// ---- POUs/EL_Terminals/FB_EL3403.TcPOU
(************************************************************************************************)
(*							Beckhoff Automation Poland											*)
(*								FB_EL3403	 v1.0												*)
(*									11.03.2014													*)
(*					Blok funkcyjny obsługujący moduł EL3403										*)
(*			Możliwy zapis energii w module, kasowanie przechowywanych wartosci					*)
(*		Jesli jest wybrany wiecej niz jeden kanal to komenda wykonana zostanie na wszystkich	*)
(*					Zapis ma wyzszy priorytet niz kasowanie										*)
(*							Blok posiada fukcje autozapisu										*)
(*				Komendy wkonywane sa na narastajace zbocze na odpowiednim wejsciu				*)
(*______________________________________________________________________________________________*)
FUNCTION_BLOCK FB_EL3403
VAR_INPUT
	sNetId					:	T_AmsNetId;							(* AMS Net ID of EtherCAT Master *)
	nSlaveAddr				:	UINT;
	bStoreCh1				:	BOOL;
	bStoreCh2				:	BOOL;
	bStoreCh3				:	BOOL;
	bStoreAll				:	BOOL;
	bAutoStore				:	BOOL;
	bDeleteCh1				:	BOOL;
	bDeleteCh2				:	BOOL;
	bDeleteCh3				:	BOOL;
	bDeleteAll				:	BOOL;
END_VAR
VAR_OUTPUT
	bBusy					:	BOOL;
	bError					:	BOOL;
	nErrorID				:	UDINT;
	bMissingZeroCrossingA 	AT %I*: 	BOOL;
	bMissingZeroCrossingB 	AT %I*:		BOOL;
	bMissingZeroCrossingC 	AT %I*: 	BOOL;
	bPhaseSequenceError		AT %I*: 	BOOL;
	rCurrent1				:	REAL; (* Unit 1 A *)
	rCurrent2				: 	REAL; (* Unit 1 A *)
	rCurrent3				: 	REAL; (* Unit 1 A *)
	rVoltage1				: 	REAL; (* Unit 1 V *)
	rVoltage2				: 	REAL; (* Unit 1 V *)
	rVoltage3				: 	REAL; (* Unit 1 V *)
	rActivePower1			: 	REAL; (* Unit 1 W *)
	rActivePower2			: 	REAL; (* Unit 1 W *)
	rActivePower3			: 	REAL; (* Unit 1 W *)
	rApparentPower1			: 	REAL; (* Unit 1 VA *)
	rApparentPower2			:	REAL; (* Unit 1 VA *)
	rApparentPower3			:	REAL; (* Unit 1 VA *)
	rReactivePower1			:	REAL; (* Unit 1 VAR *)
	rReactivePower2			:	REAL; (* Unit 1 VAR *)
	rReactivePower3			:	REAL; (* Unit 1 VAR *)
	rEnergy1				: 	REAL; (* Unit 1 Wh *)
	rEnergy2				:	REAL; (* Unit 1 Wh *)
	rEnergy3				: 	REAL; (* Unit 1 Wh *)
	rCosPhi1				: 	REAL; (* Unit 1 *)
	rCosPhi2				: 	REAL; (* Unit 1 *)
	rCosPhi3				: 	REAL; (* Unit 1 *)
	rFrequency1				: 	REAL; (* Unit 1 Hz *)
	rFrequency2				: 	REAL; (* Unit 1 Hz *)
	rFrequency3				: 	REAL; (* Unit 1 Hz *)
	rEnergyNegative1		: 	REAL; (* Unit 1 Wh *)
	rEnergyNegative2		: 	REAL; (* Unit 1 Wh *)
	rEnergyNegative3		: 	REAL; (* Unit 1 Wh *)
END_VAR
VAR
(* I/O *)
	diCurrent1 				AT %I*: DINT;(* Unit 0,000001 A *)
	diCurrent2 				AT %I*: DINT;(* Unit 0,000001 A *)
	diCurrent3 				AT %I*: DINT;(* Unit 0,000001 A *)
	diVoltage1 				AT %I*: DINT;(* Unit 0,0001 V *)
	diVoltage2 				AT %I*: DINT;(* Unit 0,0001 V *)
	diVoltage3 				AT %I*: DINT;(* Unit 0,0001 V *)
	diActivePower1 			AT %I*: DINT;(* Unit 0,01 W *)
	diActivePower2 			AT %I*: DINT;(* Unit 0,01 W *)
	diActivePower3 			AT %I*: DINT;(* Unit 0,01 W *)
	usiIndex1			 	AT %I*: USINT;
	usiIndex2			 	AT %I*: USINT;
	usiIndex3			 	AT %I*: USINT;
	diVariantValue1 		AT %I*: DINT;
	diVariantValue2 		AT %I*: DINT;
	diVariantValue3 		AT %I*: DINT;
	usiIndex1q				AT %Q*: USINT;
	usiIndex2q			 	AT %Q*: USINT;
	usiIndex3q			 	AT %Q*: USINT;
(*Raw Values*)
	diApparentPower1		: DINT; (* Unit 0,01 VA *)
	diApparentPower2		: DINT; (* Unit 0,01 VA *)
	diApparentPower3		: DINT; (* Unit 0,01 VA *)
	diReactivePower1		: DINT; (* Unit 0,01 VAR *)
	diReactivePower2		: DINT; (* Unit 0,01 VAR *)
	diReactivePower3		: DINT; (* Unit 0,01 VAR *)
	diEnergy1				: DINT;(* Unit 0,001 Wh *)
	diEnergy2				: DINT;(* Unit 0,001 Wh *)
	diEnergy3				: DINT;(* Unit 0,001 Wh *)
	diCosPhi1				: DINT;(* Unit 0,001 *)
	diCosPhi2				: DINT;(* Unit 0,001 *)
	diCosPhi3				: DINT;(* Unit 0,001 *)
	diFrequency1			: DINT;(* Unit 0,1 Hz *)
	diFrequency2			: DINT;(* Unit 0,1 Hz *)
	diFrequency3			: DINT;(* Unit 0,1 Hz *)
	diEnergyNegative1		: DINT;(* Unit 0,001 Wh *)
	diEnergyNegative2		: DINT;(* Unit 0,001 Wh *)
	diEnergyNegative3		: DINT;(* Unit 0,001 Wh *)
(* Energy store/delete *)
	fbEcCoeSdoWrite			: FB_EcCoESdoWrite;
	t1						: TON;
	arrRTrigs				: ARRAY [1..9] OF R_TRIG;
	wDataS					: WORD;
	wDataD					: WORD;
	bExecute				: BOOL;
	BStore					: BYTE; (* bit 0 - ch1, 1 - ch2, 3 - ch3, else all *)
	BDelete					: BYTE; (* bit 0 - ch1, 1 - ch2, 3 - ch3, else all *)
	bStoreCommand			: BOOL;
	bDeleteCommand			: BOOL;
	wData					: WORD;
END_VAR
VAR CONSTANT
	nSubIndex				: BYTE				:= 16#01;
	nIndex					: WORD				:= 16#FB00;
	wChannel1				: WORD				:= 16#0100;
	wChannel2				: WORD				:= 16#0200;
	wChannel3				: WORD				:= 16#0300;
	wStore					: WORD				:= 16#0014;
	wDelete					: WORD				:= 16#0004;
	tStoreInterval			: TIME				:= T#15m;
END_VAR

(* Read Variant Variable *)
A_ReadVariantVariable();

(* Scale *)
A_Scale();

(* Energy *)
BStore.0 := bStoreCh1 OR bStoreAll;
BStore.1 := bStoreCh2 OR bStoreAll;
BStore.2 := bStoreCh3 OR bStoreAll;
CASE BStore OF
1:	wDataS := wChannel1 + wStore;
2:	wDataS := wChannel2 + wStore;
4:	wDataS := wChannel3 + wStore;
ELSE
	wDataS := wStore;
END_CASE

BDelete.0 := bDeleteCh1 OR bDeleteAll;
BDelete.1 := bDeleteCh2 OR bDeleteAll;
BDelete.2 := bDeleteCh3 OR bDeleteAll;
CASE BDelete OF
1:	wDataD := wChannel1 + wDelete;
2:	wDataD := wChannel2 + wDelete;
4:	wDataD := wChannel3 + wDelete;
ELSE
	wDataD := wDelete;
END_CASE

t1(IN:= NOT t1.Q AND bAutoStore , PT:= tStoreInterval); (* Auto store *)

arrRTrigs[1](CLK:= bStoreCh1);
arrRTrigs[2](CLK:= bStoreCh2);
arrRTrigs[3](CLK:= bStoreCh3);
arrRTrigs[4](CLK:= bStoreAll);
arrRTrigs[5](CLK:= t1.Q);
arrRTrigs[6](CLK:= bDeleteCh1);
arrRTrigs[7](CLK:= bDeleteCh2);
arrRTrigs[8](CLK:= bDeleteCh3);
arrRTrigs[9](CLK:= bDeleteAll);

bStoreCommand		:= arrRTrigs[1].Q OR arrRTrigs[2].Q OR arrRTrigs[3].Q OR arrRTrigs[4].Q OR arrRTrigs[5].Q;
bDeleteCommand	:= arrRTrigs[6].Q OR arrRTrigs[7].Q OR arrRTrigs[8].Q OR arrRTrigs[9].Q;
wData				:= SEL(bDeleteCommand, wDataS, wDataD);
bExecute			:= bStoreCommand OR bDeleteCommand;




fbEcCoeSdoWrite(
	sNetId:= sNetId,
	nSlaveAddr:= nSlaveAddr,
	nSubIndex:= nSubIndex,
	nIndex:= nIndex,
	pSrcBuf:= ADR(wData),
	cbBufLen:= 2,
	bExecute:= bExecute,
	bBusy=> bBusy,
	bError=> bError,
	nErrId=> nErrorID);

ACTION A_ReadVariantVariable:
CASE usiIndex1 OF
0:
	diApparentPower1 := diVariantValue1;
	usiIndex1q := usiIndex1+1;
1:
	diReactivePower1 := diVariantValue1;
	usiIndex1q := usiIndex1+1;
2:
	diEnergy1 := diVariantValue1;
	usiIndex1q := usiIndex1+1;
3:
	diCosPhi1 := diVariantValue1;
	usiIndex1q := usiIndex1+1;
4:
	diFrequency1 := diVariantValue1;
	usiIndex1q := usiIndex1+1;
5:
	diEnergyNegative1 := diVariantValue1;
	usiIndex1q := usiIndex1+1;
ELSE
	usiIndex1q := 0;
END_CASE

CASE usiIndex2 OF
0:
	diApparentPower2 := diVariantValue2;
	usiIndex2q := usiIndex2+1;
1:
	diReactivePower2 := diVariantValue2;
	usiIndex2q := usiIndex2+1;
2:
	diEnergy2 := diVariantValue2;
	usiIndex2q := usiIndex2+1;
3:
	diCosPhi2 := diVariantValue2;
	usiIndex2q := usiIndex2+1;
4:
	diFrequency2 := diVariantValue2;
	usiIndex2q := usiIndex2+1;
5:
	diEnergyNegative2 := diVariantValue2;
	usiIndex2q := usiIndex2+1;
ELSE
	usiIndex2q := 0;
END_CASE


CASE usiIndex3 OF
0:
	diApparentPower3 := diVariantValue3;
	usiIndex3q := usiIndex3+1;
1:
	diReactivePower3 := diVariantValue3;
	usiIndex3q := usiIndex3+1;
2:
	diEnergy3 := diVariantValue3;
	usiIndex3q := usiIndex3+1;
3:
	diCosPhi3 := diVariantValue3;
	usiIndex3q := usiIndex3+1;
4:
	diFrequency3 := diVariantValue3;
	usiIndex3q := usiIndex3+1;
5:
	diEnergyNegative3 := diVariantValue3;
	usiIndex3q := usiIndex3+1;
ELSE
	usiIndex3q := 0;
END_CASE
END_ACTION

ACTION A_Scale:
	rCurrent1 			:= DINT_TO_REAL(diCurrent1)*0.000001;
	rVoltage1 			:= DINT_TO_REAL(diVoltage1)*0.0001;
	rActivePower1	 	:= DINT_TO_REAL(diActivePower1)*0.01;
	rApparentPower1 	:= DINT_TO_REAL(diApparentPower1)*0.01;
	rReactivePower1 	:= DINT_TO_REAL(diReactivePower1)*0.01;
	rEnergy1 			:= DINT_TO_REAL(diEnergy1)*0.0001;
	rCosPhi1 			:= DINT_TO_REAL(diCosPhi1)*0.001;
	rFrequency1 		:= DINT_TO_REAL(diFrequency1)*0.1;
	rEnergyNegative1 	:= DINT_TO_REAL(diEnergyNegative1)*0.001;

	rCurrent2 			:= DINT_TO_REAL(diCurrent2)*0.000001;
	rVoltage2 			:= DINT_TO_REAL(diVoltage2)*0.0001;
	rActivePower2	 	:= DINT_TO_REAL(diActivePower2)*0.01;
	rApparentPower2 	:= DINT_TO_REAL(diApparentPower2)*0.01;
	rReactivePower2 	:= DINT_TO_REAL(diReactivePower2)*0.01;
	rEnergy2 			:= DINT_TO_REAL(diEnergy2)*0.0001;
	rCosPhi2 			:= DINT_TO_REAL(diCosPhi2)*0.001;
	rFrequency2 		:= DINT_TO_REAL(diFrequency2)*0.1;
	rEnergyNegative2 	:= DINT_TO_REAL(diEnergyNegative2)*0.001;

	rCurrent3 			:= DINT_TO_REAL(diCurrent3)*0.000001;
	rVoltage3 			:= DINT_TO_REAL(diVoltage3)*0.0001;
	rActivePower3	 	:= DINT_TO_REAL(diActivePower3)*0.01;
	rApparentPower3 	:= DINT_TO_REAL(diApparentPower3)*0.01;
	rReactivePower3 	:= DINT_TO_REAL(diReactivePower3)*0.01;
	rEnergy3 			:= DINT_TO_REAL(diEnergy3)*0.0001;
	rCosPhi3 			:= DINT_TO_REAL(diCosPhi3)*0.001;
	rFrequency3 		:= DINT_TO_REAL(diFrequency3)*0.1;
	rEnergyNegative3 	:= DINT_TO_REAL(diEnergyNegative3)*0.001;
END_ACTION

END_FUNCTION_BLOCK

// ---- POUs/EL_Terminals/FB_EL3403Ex.TcPOU
(************************************************************************************************)
(*							Beckhoff Automation Poland											*)
(*								FB_EL3403Ex	 v1.0												*)
(*									11.03.2014													*)
(*					Blok funkcyjny obsługujący moduł EL3403										*)
(*			Możliwy zapis energii w module, kasowanie przechowywanych wartosci					*)
(*		Jesli jest wybrany wiecej niz jeden kanal to komenda wykonana zostanie na wszystkich	*)
(*					Zapis ma wyzszy priorytet niz kasowanie										*)
(*							Blok posiada fukcje autozapisu										*)
(*				Komendy wkonywane sa na narastajace zbocze na odpowiednim wejsciu				*)
(* 				Wyjscia z danymi udostepniopne w formie struktury ST_EL3403_Data 				*)
(*______________________________________________________________________________________________*)
FUNCTION_BLOCK FB_EL3403Ex
VAR_INPUT
	sNetId					: T_AmsNetId; (* AMS Net ID of EtherCAT Master *)
	nSlaveAddr				: UINT;
	bStoreCh1				: BOOL;
	bStoreCh2				: BOOL;
	bStoreCh3				: BOOL;
	bStoreAll				: BOOL;
	bAutoStore				: BOOL;
	bDeleteCh1				: BOOL;
	bDeleteCh2				: BOOL;
	bDeleteCh3				: BOOL;
	bDeleteAll				: BOOL;
END_VAR
VAR_OUTPUT
	bBusy					: BOOL;
	bError					: BOOL;
	nErrorID				: UDINT;
	bMissingZeroCrossingA 	AT %I*: BOOL;
	bMissingZeroCrossingB 	AT %I*: BOOL;
	bMissingZeroCrossingC 	AT %I*: BOOL;
	bPhaseSequenceError		AT %I*: BOOL;
	stEL3403_Data			:ST_EL3403_Data; (*Parametry wyjściowe*)
END_VAR
VAR
(* I/O *)
	diCurrent1 				AT %I*: DINT;(* Unit 0,000001 A *)
	diCurrent2 				AT %I*: DINT;(* Unit 0,000001 A *)
	diCurrent3 				AT %I*: DINT;(* Unit 0,000001 A *)
	diVoltage1 				AT %I*: DINT;(* Unit 0,0001 V *)
	diVoltage2 				AT %I*: DINT;(* Unit 0,0001 V *)
	diVoltage3 				AT %I*: DINT;(* Unit 0,0001 V *)
	diActivePower1 			AT %I*: DINT;(* Unit 0,01 W *)
	diActivePower2 			AT %I*: DINT;(* Unit 0,01 W *)
	diActivePower3 			AT %I*: DINT;(* Unit 0,01 W *)
	usiIndex1				AT %I*: USINT;
	usiIndex2				AT %I*: USINT;
	usiIndex3				AT %I*: USINT;
	diVariantValue1 		AT %I*: DINT;
	diVariantValue2 		AT %I*: DINT;
	diVariantValue3 		AT %I*: DINT;
	usiIndex1q				AT %Q*: USINT;
	usiIndex2q				AT %Q*: USINT;
	usiIndex3q				AT %Q*: USINT;
(*Raw Values*)
	diApparentPower1		: DINT; (* Unit 0,01 VA *)
	diApparentPower2		: DINT; (* Unit 0,01 VA *)
	diApparentPower3		: DINT; (* Unit 0,01 VA *)
	diReactivePower1		: DINT; (* Unit 0,01 VAR *)
	diReactivePower2		: DINT; (* Unit 0,01 VAR *)
	diReactivePower3		: DINT; (* Unit 0,01 VAR *)
	diEnergy1				: DINT;(* Unit 0,001 Wh *)
	diEnergy2				: DINT;(* Unit 0,001 Wh *)
	diEnergy3				: DINT;(* Unit 0,001 Wh *)
	diCosPhi1				: DINT;(* Unit 0,001 *)
	diCosPhi2				: DINT;(* Unit 0,001 *)
	diCosPhi3				: DINT;(* Unit 0,001 *)
	diFrequency1			: DINT;(* Unit 0,1 Hz *)
	diFrequency2			: DINT;(* Unit 0,1 Hz *)
	diFrequency3			: DINT;(* Unit 0,1 Hz *)
	diEnergyNegative1		: DINT;(* Unit 0,001 Wh *)
	diEnergyNegative2		: DINT;(* Unit 0,001 Wh *)
	diEnergyNegative3		: DINT;(* Unit 0,001 Wh *)
(* Energy store/delete *)
	fbEcCoeSdoWrite			: FB_EcCoESdoWrite;
	t1						: TON;
	arrRTrigs				: ARRAY [1..9] OF R_TRIG;
	wDataS					: WORD;
	wDataD					: WORD;
	bExecute				: BOOL;
	BStore					: BYTE; (* bit 0 - ch1, 1 - ch2, 3 - ch3, else all *)
	BDelete					: BYTE; (* bit 0 - ch1, 1 - ch2, 3 - ch3, else all *)
	bStoreCommand			: BOOL;
	bDeleteCommand			: BOOL;
	wData					: WORD;

END_VAR
VAR CONSTANT
	nSubIndex				: BYTE				:= 16#01;
	nIndex					: WORD				:= 16#FB00;
	wChannel1				: WORD				:= 16#0100;
	wChannel2				: WORD				:= 16#0200;
	wChannel3				: WORD				:= 16#0300;
	wStore					: WORD				:= 16#0014;
	wDelete					: WORD				:= 16#0004;
	tStoreInterval			: TIME				:= T#15m;
END_VAR

(* Read Variant Variable *)
A_ReadVariantVariable();

(* Scale *)
A_Scale();

(* Energy *)
BStore.0 := bStoreCh1 OR bStoreAll;
BStore.1 := bStoreCh2 OR bStoreAll;
BStore.2 := bStoreCh3 OR bStoreAll;
CASE BStore OF
1:	wDataS := wChannel1 + wStore;
2:	wDataS := wChannel2 + wStore;
4:	wDataS := wChannel3 + wStore;
ELSE
	wDataS := wStore;
END_CASE

BDelete.0 := bDeleteCh1 OR bDeleteAll;
BDelete.1 := bDeleteCh2 OR bDeleteAll;
BDelete.2 := bDeleteCh3 OR bDeleteAll;
CASE BDelete OF
1:	wDataD := wChannel1 + wDelete;
2:	wDataD := wChannel2 + wDelete;
4:	wDataD := wChannel3 + wDelete;
ELSE
	wDataD := wDelete;
END_CASE

t1(IN:= NOT t1.Q AND bAutoStore , PT:= tStoreInterval); (* Auto store *)

arrRTrigs[1](CLK:= bStoreCh1);
arrRTrigs[2](CLK:= bStoreCh2);
arrRTrigs[3](CLK:= bStoreCh3);
arrRTrigs[4](CLK:= bStoreAll);
arrRTrigs[5](CLK:= t1.Q);
arrRTrigs[6](CLK:= bDeleteCh1);
arrRTrigs[7](CLK:= bDeleteCh2);
arrRTrigs[8](CLK:= bDeleteCh3);
arrRTrigs[9](CLK:= bDeleteAll);

bStoreCommand		:= arrRTrigs[1].Q OR arrRTrigs[2].Q OR arrRTrigs[3].Q OR arrRTrigs[4].Q OR arrRTrigs[5].Q;
bDeleteCommand	:= arrRTrigs[6].Q OR arrRTrigs[7].Q OR arrRTrigs[8].Q OR arrRTrigs[9].Q;
wData				:= SEL(bDeleteCommand, wDataS, wDataD);
bExecute			:= bStoreCommand OR bDeleteCommand;




fbEcCoeSdoWrite(
	sNetId:= sNetId,
	nSlaveAddr:= nSlaveAddr,
	nSubIndex:= nSubIndex,
	nIndex:= nIndex,
	pSrcBuf:= ADR(wData),
	cbBufLen:= 2,
	bExecute:= bExecute,
	bBusy=> bBusy,
	bError=> bError,
	nErrId=> nErrorID);

ACTION A_ReadVariantVariable:
CASE usiIndex1 OF
0:
	diApparentPower1 := diVariantValue1;
	usiIndex1q := usiIndex1+1;
1:
	diReactivePower1 := diVariantValue1;
	usiIndex1q := usiIndex1+1;
2:
	diEnergy1 := diVariantValue1;
	usiIndex1q := usiIndex1+1;
3:
	diCosPhi1 := diVariantValue1;
	usiIndex1q := usiIndex1+1;
4:
	diFrequency1 := diVariantValue1;
	usiIndex1q := usiIndex1+1;
5:
	diEnergyNegative1 := diVariantValue1;
	usiIndex1q := usiIndex1+1;
ELSE
	usiIndex1q := 0;
END_CASE

CASE usiIndex2 OF
0:
	diApparentPower2 := diVariantValue2;
	usiIndex2q := usiIndex2+1;
1:
	diReactivePower2 := diVariantValue2;
	usiIndex2q := usiIndex2+1;
2:
	diEnergy2 := diVariantValue2;
	usiIndex2q := usiIndex2+1;
3:
	diCosPhi2 := diVariantValue2;
	usiIndex2q := usiIndex2+1;
4:
	diFrequency2 := diVariantValue2;
	usiIndex2q := usiIndex2+1;
5:
	diEnergyNegative2 := diVariantValue2;
	usiIndex2q := usiIndex2+1;
ELSE
	usiIndex2q := 0;
END_CASE


CASE usiIndex3 OF
0:
	diApparentPower3 := diVariantValue3;
	usiIndex3q := usiIndex3+1;
1:
	diReactivePower3 := diVariantValue3;
	usiIndex3q := usiIndex3+1;
2:
	diEnergy3 := diVariantValue3;
	usiIndex3q := usiIndex3+1;
3:
	diCosPhi3 := diVariantValue3;
	usiIndex3q := usiIndex3+1;
4:
	diFrequency3 := diVariantValue3;
	usiIndex3q := usiIndex3+1;
5:
	diEnergyNegative3 := diVariantValue3;
	usiIndex3q := usiIndex3+1;
ELSE
	usiIndex3q := 0;
END_CASE
END_ACTION

ACTION A_Scale:
	stEL3403_Data.rCurrent1 			:= DINT_TO_REAL(diCurrent1)*0.000001;
	stEL3403_Data.rVoltage1 			:= DINT_TO_REAL(diVoltage1)*0.0001;
	stEL3403_Data.rActivePower1	 		:= DINT_TO_REAL(diActivePower1)*0.01;
	stEL3403_Data.rApparentPower1	 	:= DINT_TO_REAL(diApparentPower1)*0.01;
	stEL3403_Data.rReactivePower1 		:= DINT_TO_REAL(diReactivePower1)*0.01;
	stEL3403_Data.rEnergy1 				:= DINT_TO_REAL(diEnergy1)*0.0001;
	stEL3403_Data.rCosPhi1	 			:= DINT_TO_REAL(diCosPhi1)*0.001;
	stEL3403_Data.rFrequency1	 		:= DINT_TO_REAL(diFrequency1)*0.1;
	stEL3403_Data.rEnergyNegative1	 	:= DINT_TO_REAL(diEnergyNegative1)*0.001;

	stEL3403_Data.rCurrent2 			:= DINT_TO_REAL(diCurrent2)*0.000001;
	stEL3403_Data.rVoltage2 			:= DINT_TO_REAL(diVoltage2)*0.0001;
	stEL3403_Data.rActivePower2	 		:= DINT_TO_REAL(diActivePower2)*0.01;
	stEL3403_Data.rApparentPower2 		:= DINT_TO_REAL(diApparentPower2)*0.01;
	stEL3403_Data.rReactivePower2	 	:= DINT_TO_REAL(diReactivePower2)*0.01;
	stEL3403_Data.rEnergy2 				:= DINT_TO_REAL(diEnergy2)*0.0001;
	stEL3403_Data.rCosPhi2	 			:= DINT_TO_REAL(diCosPhi2)*0.001;
	stEL3403_Data.rFrequency2	 		:= DINT_TO_REAL(diFrequency2)*0.1;
	stEL3403_Data.rEnergyNegative2 		:= DINT_TO_REAL(diEnergyNegative2)*0.001;

	stEL3403_Data.rCurrent3 			:= DINT_TO_REAL(diCurrent3)*0.000001;
	stEL3403_Data.rVoltage3 			:= DINT_TO_REAL(diVoltage3)*0.0001;
	stEL3403_Data.rActivePower3	 		:= DINT_TO_REAL(diActivePower3)*0.01;
	stEL3403_Data.rApparentPower3 		:= DINT_TO_REAL(diApparentPower3)*0.01;
	stEL3403_Data.rReactivePower3 		:= DINT_TO_REAL(diReactivePower3)*0.01;
	stEL3403_Data.rEnergy3 				:= DINT_TO_REAL(diEnergy3)*0.0001;
	stEL3403_Data.rCosPhi3 				:= DINT_TO_REAL(diCosPhi3)*0.001;
	stEL3403_Data.rFrequency3 			:= DINT_TO_REAL(diFrequency3)*0.1;
	stEL3403_Data.rEnergyNegative3 		:= DINT_TO_REAL(diEnergyNegative3)*0.001;
END_ACTION

END_FUNCTION_BLOCK

// ---- POUs/EL_Terminals/FB_EL3403Ex2.TcPOU
(************************************************************************************************)
(*							Beckhoff Automation Poland											*)
(*								FB_EL3403Ex2	 v1.0											*)
(*									26.02.2015													*)
(*					Blok funkcyjny obsługujący moduł EL3403										*)
(*				Roznica w porownaniu z FB_EL3403Ex - mozliwe dodanie							*)
(*				wartosci przekladnikow pradowych dla kazdego kanalu 							*)
(*			Możliwy zapis energii w module, kasowanie przechowywanych wartosci					*)
(*		Jesli jest wybrany wiecej niz jeden kanal to komenda wykonana zostanie na wszystkich	*)
(*					Zapis ma wyzszy priorytet niz kasowanie										*)
(*							Blok posiada fukcje autozapisu										*)
(*				Komendy wkonywane sa na narastajace zbocze na odpowiednim wejsciu				*)
(* 				Wyjscia z danymi udostepniopne w formie struktury ST_EL3403_Data 				*)
(*______________________________________________________________________________________________*)
FUNCTION_BLOCK FB_EL3403Ex2
VAR_INPUT
	sNetId					: T_AmsNetId; (* AMS Net ID of EtherCAT Master *)
	nSlaveAddr				: UINT;
	bStoreCh1				: BOOL;
	bStoreCh2				: BOOL;
	bStoreCh3				: BOOL;
	bStoreAll				: BOOL;
	bAutoStore				: BOOL;
	bDeleteCh1				: BOOL;
	bDeleteCh2				: BOOL;
	bDeleteCh3				: BOOL;
	bDeleteAll				: BOOL;
	rCurrentTransformer1	: REAL := 1.0;
	rCurrentTransformer2	: REAL := 1.0;
	rCurrentTransformer3	: REAL := 1.0;
END_VAR
VAR_OUTPUT
	bBusy					: BOOL;
	bError					: BOOL;
	nErrorID				: UDINT;
	bMissingZeroCrossingA 	AT %I*: BOOL;
	bMissingZeroCrossingB 	AT %I*: BOOL;
	bMissingZeroCrossingC 	AT %I*: BOOL;
	bPhaseSequenceError		AT %I*: BOOL;
	stEL3403_Data			:ST_EL3403_Data; (*Parametry wyjściowe*)
END_VAR
VAR
(* I/O *)
	diCurrent1 				AT %I*: DINT;(* Unit 0,000001 A *)
	diCurrent2 				AT %I*: DINT;(* Unit 0,000001 A *)
	diCurrent3 				AT %I*: DINT;(* Unit 0,000001 A *)
	diVoltage1 				AT %I*: DINT;(* Unit 0,0001 V *)
	diVoltage2 				AT %I*: DINT;(* Unit 0,0001 V *)
	diVoltage3 				AT %I*: DINT;(* Unit 0,0001 V *)
	diActivePower1 			AT %I*: DINT;(* Unit 0,01 W *)
	diActivePower2 			AT %I*: DINT;(* Unit 0,01 W *)
	diActivePower3 			AT %I*: DINT;(* Unit 0,01 W *)
	usiIndex1				AT %I*: USINT;
	usiIndex2				AT %I*: USINT;
	usiIndex3				AT %I*: USINT;
	diVariantValue1 		AT %I*: DINT;
	diVariantValue2 		AT %I*: DINT;
	diVariantValue3 		AT %I*: DINT;
	usiIndex1q				AT %Q*: USINT;
	usiIndex2q				AT %Q*: USINT;
	usiIndex3q				AT %Q*: USINT;
(*Raw Values*)
	diApparentPower1		: DINT; (* Unit 0,01 VA *)
	diApparentPower2		: DINT; (* Unit 0,01 VA *)
	diApparentPower3		: DINT; (* Unit 0,01 VA *)
	diReactivePower1		: DINT; (* Unit 0,01 VAR *)
	diReactivePower2		: DINT; (* Unit 0,01 VAR *)
	diReactivePower3		: DINT; (* Unit 0,01 VAR *)
	diEnergy1				: DINT;(* Unit 0,001 Wh *)
	diEnergy2				: DINT;(* Unit 0,001 Wh *)
	diEnergy3				: DINT;(* Unit 0,001 Wh *)
	diCosPhi1				: DINT;(* Unit 0,001 *)
	diCosPhi2				: DINT;(* Unit 0,001 *)
	diCosPhi3				: DINT;(* Unit 0,001 *)
	diFrequency1			: DINT;(* Unit 0,1 Hz *)
	diFrequency2			: DINT;(* Unit 0,1 Hz *)
	diFrequency3			: DINT;(* Unit 0,1 Hz *)
	diEnergyNegative1		: DINT;(* Unit 0,001 Wh *)
	diEnergyNegative2		: DINT;(* Unit 0,001 Wh *)
	diEnergyNegative3		: DINT;(* Unit 0,001 Wh *)
(* Energy store/delete *)
	fbEcCoeSdoWrite			: FB_EcCoESdoWrite;
	t1						: TON;
	arrRTrigs				: ARRAY [1..9] OF R_TRIG;
	wDataS					: WORD;
	wDataD					: WORD;
	bExecute				: BOOL;
	BStore					: BYTE; (* bit 0 - ch1, 1 - ch2, 3 - ch3, else all *)
	BDelete					: BYTE; (* bit 0 - ch1, 1 - ch2, 3 - ch3, else all *)
	bStoreCommand			: BOOL;
	bDeleteCommand			: BOOL;
	wData					: WORD;

END_VAR
VAR CONSTANT
	nSubIndex				: BYTE				:= 16#01;
	nIndex					: WORD				:= 16#FB00;
	wChannel1				: WORD				:= 16#0100;
	wChannel2				: WORD				:= 16#0200;
	wChannel3				: WORD				:= 16#0300;
	wStore					: WORD				:= 16#0014;
	wDelete					: WORD				:= 16#0004;
	tStoreInterval			: TIME				:= T#15m;
END_VAR

(* Read Variant Variable *)
A_ReadVariantVariable();

(* Scale *)
A_Scale();

(* Energy *)
BStore.0 := bStoreCh1 OR bStoreAll;
BStore.1 := bStoreCh2 OR bStoreAll;
BStore.2 := bStoreCh3 OR bStoreAll;
CASE BStore OF
1:	wDataS := wChannel1 + wStore;
2:	wDataS := wChannel2 + wStore;
4:	wDataS := wChannel3 + wStore;
ELSE
	wDataS := wStore;
END_CASE

BDelete.0 := bDeleteCh1 OR bDeleteAll;
BDelete.1 := bDeleteCh2 OR bDeleteAll;
BDelete.2 := bDeleteCh3 OR bDeleteAll;
CASE BDelete OF
1:	wDataD := wChannel1 + wDelete;
2:	wDataD := wChannel2 + wDelete;
4:	wDataD := wChannel3 + wDelete;
ELSE
	wDataD := wDelete;
END_CASE

t1(IN:= NOT t1.Q AND bAutoStore , PT:= tStoreInterval); (* Auto store *)

arrRTrigs[1](CLK:= bStoreCh1);
arrRTrigs[2](CLK:= bStoreCh2);
arrRTrigs[3](CLK:= bStoreCh3);
arrRTrigs[4](CLK:= bStoreAll);
arrRTrigs[5](CLK:= t1.Q);
arrRTrigs[6](CLK:= bDeleteCh1);
arrRTrigs[7](CLK:= bDeleteCh2);
arrRTrigs[8](CLK:= bDeleteCh3);
arrRTrigs[9](CLK:= bDeleteAll);

bStoreCommand		:= arrRTrigs[1].Q OR arrRTrigs[2].Q OR arrRTrigs[3].Q OR arrRTrigs[4].Q OR arrRTrigs[5].Q;
bDeleteCommand	:= arrRTrigs[6].Q OR arrRTrigs[7].Q OR arrRTrigs[8].Q OR arrRTrigs[9].Q;
wData				:= SEL(bDeleteCommand, wDataS, wDataD);
bExecute			:= bStoreCommand OR bDeleteCommand;




fbEcCoeSdoWrite(
	sNetId:= sNetId,
	nSlaveAddr:= nSlaveAddr,
	nSubIndex:= nSubIndex,
	nIndex:= nIndex,
	pSrcBuf:= ADR(wData),
	cbBufLen:= 2,
	bExecute:= bExecute,
	bBusy=> bBusy,
	bError=> bError,
	nErrId=> nErrorID);

ACTION A_ReadVariantVariable:
CASE usiIndex1 OF
0:
	diApparentPower1 := diVariantValue1;
	usiIndex1q := usiIndex1+1;
1:
	diReactivePower1 := diVariantValue1;
	usiIndex1q := usiIndex1+1;
2:
	diEnergy1 := diVariantValue1;
	usiIndex1q := usiIndex1+1;
3:
	diCosPhi1 := diVariantValue1;
	usiIndex1q := usiIndex1+1;
4:
	diFrequency1 := diVariantValue1;
	usiIndex1q := usiIndex1+1;
5:
	diEnergyNegative1 := diVariantValue1;
	usiIndex1q := usiIndex1+1;
ELSE
	usiIndex1q := 0;
END_CASE

CASE usiIndex2 OF
0:
	diApparentPower2 := diVariantValue2;
	usiIndex2q := usiIndex2+1;
1:
	diReactivePower2 := diVariantValue2;
	usiIndex2q := usiIndex2+1;
2:
	diEnergy2 := diVariantValue2;
	usiIndex2q := usiIndex2+1;
3:
	diCosPhi2 := diVariantValue2;
	usiIndex2q := usiIndex2+1;
4:
	diFrequency2 := diVariantValue2;
	usiIndex2q := usiIndex2+1;
5:
	diEnergyNegative2 := diVariantValue2;
	usiIndex2q := usiIndex2+1;
ELSE
	usiIndex2q := 0;
END_CASE


CASE usiIndex3 OF
0:
	diApparentPower3 := diVariantValue3;
	usiIndex3q := usiIndex3+1;
1:
	diReactivePower3 := diVariantValue3;
	usiIndex3q := usiIndex3+1;
2:
	diEnergy3 := diVariantValue3;
	usiIndex3q := usiIndex3+1;
3:
	diCosPhi3 := diVariantValue3;
	usiIndex3q := usiIndex3+1;
4:
	diFrequency3 := diVariantValue3;
	usiIndex3q := usiIndex3+1;
5:
	diEnergyNegative3 := diVariantValue3;
	usiIndex3q := usiIndex3+1;
ELSE
	usiIndex3q := 0;
END_CASE
END_ACTION

ACTION A_Scale:
	stEL3403_Data.rCurrent1 			:= DINT_TO_REAL(diCurrent1)*0.000001*rCurrentTransformer1; (**)
	stEL3403_Data.rVoltage1 			:= DINT_TO_REAL(diVoltage1)*0.0001;
	stEL3403_Data.rActivePower1	 		:= DINT_TO_REAL(diActivePower1)*0.01*rCurrentTransformer1; (**)
	stEL3403_Data.rApparentPower1 		:= DINT_TO_REAL(diApparentPower1)*0.01*rCurrentTransformer1; (**)
	stEL3403_Data.rReactivePower1 		:= DINT_TO_REAL(diReactivePower1)*0.01*rCurrentTransformer1; (**)
	stEL3403_Data.rEnergy1 				:= DINT_TO_REAL(diEnergy1)*0.0001*rCurrentTransformer1; (**)
	stEL3403_Data.rCosPhi1 				:= DINT_TO_REAL(diCosPhi1)*0.001;
	stEL3403_Data.rFrequency1 			:= DINT_TO_REAL(diFrequency1)*0.1;
	stEL3403_Data.rEnergyNegative1 		:= DINT_TO_REAL(diEnergyNegative1)*0.001*rCurrentTransformer1; (**)

	stEL3403_Data.rCurrent2 			:= DINT_TO_REAL(diCurrent2)*0.000001*rCurrentTransformer2; (**)
	stEL3403_Data.rVoltage2 			:= DINT_TO_REAL(diVoltage2)*0.0001;
	stEL3403_Data.rActivePower2	 		:= DINT_TO_REAL(diActivePower2)*0.01*rCurrentTransformer2; (**)
	stEL3403_Data.rApparentPower2 		:= DINT_TO_REAL(diApparentPower2)*0.01*rCurrentTransformer2; (**)
	stEL3403_Data.rReactivePower2 		:= DINT_TO_REAL(diReactivePower2)*0.01*rCurrentTransformer2; (**)
	stEL3403_Data.rEnergy2 				:= DINT_TO_REAL(diEnergy2)*0.0001*rCurrentTransformer2; (**)
	stEL3403_Data.rCosPhi2 				:= DINT_TO_REAL(diCosPhi2)*0.001;
	stEL3403_Data.rFrequency2 			:= DINT_TO_REAL(diFrequency2)*0.1;
	stEL3403_Data.rEnergyNegative2 		:= DINT_TO_REAL(diEnergyNegative2)*0.001*rCurrentTransformer2; (**)

	stEL3403_Data.rCurrent3 			:= DINT_TO_REAL(diCurrent3)*0.000001*rCurrentTransformer3; (**)
	stEL3403_Data.rVoltage3 			:= DINT_TO_REAL(diVoltage3)*0.0001;
	stEL3403_Data.rActivePower3	 		:= DINT_TO_REAL(diActivePower3)*0.01*rCurrentTransformer3; (**)
	stEL3403_Data.rApparentPower3 		:= DINT_TO_REAL(diApparentPower3)*0.01*rCurrentTransformer3; (**)
	stEL3403_Data.rReactivePower3 		:= DINT_TO_REAL(diReactivePower3)*0.01*rCurrentTransformer3; (**)
	stEL3403_Data.rEnergy3 				:= DINT_TO_REAL(diEnergy3)*0.0001*rCurrentTransformer3; (**)
	stEL3403_Data.rCosPhi3 				:= DINT_TO_REAL(diCosPhi3)*0.001;
	stEL3403_Data.rFrequency3 			:= DINT_TO_REAL(diFrequency3)*0.1;
	stEL3403_Data.rEnergyNegative3 		:= DINT_TO_REAL(diEnergyNegative3)*0.001*rCurrentTransformer3; (**)
END_ACTION

END_FUNCTION_BLOCK

// ---- POUs/FileAccess/FB_EmailLog.TcPOU
(****************************************************************************************)
(*							Beckhoff Automation Poland									*)
(*								FB_EmailLog  v2.0										*)
(*									26.06.2014											*)
(*			v2.0 - zmiana układu wejsc, zapis zmiennej STRING(1000)						*)
(*			Blok funkcyjny pozwalający logowac dane poprzez e-mail						*)
(*						wymaga biblioteki TcSmtp.lib									*)
(*	Uwaga - blok nie posiada reakcji na zbocze narastajace,								*)
(*	aby mogl byc wykorzystany wielokrotnie w jednym cyklu programu. 					*)
(*	Reakcja na zbocze musi byc wykonana na zewnatrz bloku. 								*)
(*	W przypadku pojawiania sie komunikatow czesciej niz blok jest w stanie wyslac,		*)
(*	dane sa buforowane w pamieci w zmiennej arrSMTPBuffer: ARRAY [1..4] OF STRING; 		*)
(*______________________________________________________________________________________*)
FUNCTION_BLOCK FB_EmailLog
VAR_INPUT
	bAdd					: BOOL;			(* Dodaj wpis *)
	sMessage				: STRING;		(* Tresc wpisu *)
	bNoAndTime				: BOOL:= TRUE; (* TRUE - dodaj nr porzadkowy i stempel czasowy *)
	sActTime				: STRING;		(* Aktualny czas *)
(* Ustawienia serwera *)
	AmsNetId				: T_AmsNetId;	(* AMS NET ID obiektu docelowego, gdy lokalnie, to zmienna moze byc pusta *)
	sSmtpServer				: STRING;
	sUsername				: STRING;
	sPassword				: STRING;
	sFrom					: STRING;
	sTo						: STRING;
	sCc						: STRING;
	sBcc					: STRING;
	sSubject				: STRING;

END_VAR
VAR_OUTPUT
	bBusy					: BOOL;
	bError					: BOOL;
END_VAR
VAR
(* Wysyłanie maila *)
	fbSMTPv3: 				FB_SmtpV3;
	fbSMTPBuffer:			FB_StringRingBuffer;
	arrSMTPBuffer:	 		ARRAY [1..4] OF STRING;
	wMessageNo: 			WORD;
	sEMailMessage: 			STRING;
	nStep: 					BYTE;
END_VAR

fbSMTPBuffer(pBuffer:= ADR(arrSMTPBuffer),
			cbBuffer:= SIZEOF(arrSMTPBuffer));

IF bAdd THEN
	IF bNoAndTime THEN
		wMessageNo:=wMessageNo + 1;
		sMessage := CONCAT(CONCAT(CONCAT(CONCAT(CONCAT(WORD_TO_STRING(wMessageNo),'.$t'),sActTime),'$t'),sMessage),'$n');
	END_IF
	fbSMTPBuffer.A_AddTail(putValue:= sMessage);
END_IF

CASE nStep OF
	0:
	(* Jesli jest komunikat do wyslania to wyslij *)
	IF fbSMTPBuffer.nCount>0 THEN
		fbSMTPBuffer.A_RemoveHead(getValue=> sEMailMessage);
		fbSMTPv3.bExecute:=TRUE;
		nStep := nStep + 10;
	END_IF
	10:
	fbSMTPv3.bExecute:=FALSE;
	(* Jak wyslanie zakonczone sukcesem - to wroc do kroku 0 *)
	IF NOT bBusy AND NOT bError THEN
		nStep := 0;
	END_IF
	(* Jak blad to zresetuj bloczek i podejmij próbę ponownie *)
	IF bError THEN
		nStep := nStep + 10;
	END_IF
	20:
		fbSMTPv3.bExecute:=TRUE;
		nStep := nStep - 10;
END_CASE

fbSMTPv3(
	sNetId			:= AmsNetId,
	sSmtpServer		:= sSmtpServer,
	sUsername		:= sUsername,
	sPassword		:= sPassword,
	nEncryption     := 2,
	sFrom			:= sFrom,
	sTo				:= sTo,
	sCc				:= sCc,
	sBcc			:= sBcc,
	sSubject		:= sSubject,
	pMessage		:= ADR(sEMailMessage),
	cbMessage		:= SIZEOF(sEMailMessage),
	bBusy			=> bBusy,
	bError			=> bError);

END_FUNCTION_BLOCK

// ---- POUs/FileAccess/FB_FileLog.TcPOU
(****************************************************************************************)
(*							Beckhoff Automation Poland									*)
(*								FB_FileLog  v1.0										*)
(*									26.06.2014											*)
(*			Blok funkcyjny pozwalający logowac dane do pliku							*)
(*	Uwaga - blok nie posiada reakcji na zbocze narastajace,								*)
(*	aby mogl byc wykorzystany wielokrotnie w jednym cyklu programu. 					*)
(*	Reakcja na zbocze musi byc wykonana na zewnatrz bloku. 								*)
(*	W przypadku pojawiania sie komunikatow czesciej niz blok jest w stanie zapisac,		*)
(*	dane sa buforowane w pamieci w zmiennej 											*)
 (*	arrSaveEventBuffer:ARRAY [1..20] OF STRING; 										*)
(*______________________________________________________________________________________*)
FUNCTION_BLOCK FB_FileLog
VAR_INPUT
	bAdd					: BOOL;			(* Dodaj wpis *)
	sMessage				: STRING(1000);	(* Tresc wpisu *)
	bNoAndTime				: BOOL:= TRUE; (* TRUE - dodaj nr porzadkowy i stempel czasowy *)
	sActTime				: STRING;		(* Aktualny czas *)
(* Ustawienia zapisu do pliku *)
	AmsNetId				: T_AmsNetId;	(* AMS NET ID obiektu docelowego, gdy lokalnie, to zmienna moze byc pusta *)
	sPath					: STRING; 		(* Sciezka pliku, np  'Hard Disk\'*)
	sName					: STRING; 		(* Nazwa pliku wraz z rozszerzeniem 'LogFile.txt'; *)
END_VAR
VAR_OUTPUT
	bBusy					: BOOL;
	bError					: BOOL;
END_VAR
VAR
(* Logowanie do plików *)
	fbSaveEvent: 			FB_SaveTextToFile;
	fbSaveEventBuffer:		FB_MemRingBuffer;
	arrSaveEventBuffer: 	ARRAY [1..20] OF STRING(1000);
	wMessageNo: 			WORD;
	sFileMessage: 			STRING(1000);
	nStep: 					BYTE;
END_VAR

fbSaveEventBuffer(
	pWrite:= ADR(sMessage),
	cbWrite:= SIZEOF(sMessage),
	pRead:= ADR(sFileMessage),
	cbRead:= SIZEOF(sFileMessage),
	pBuffer:= ADR(arrSaveEventBuffer),
	cbBuffer:= SIZEOF(arrSaveEventBuffer),
	bOk=> ,
	nCount=> , 
	cbSize=> , 
	cbReturn=> );
IF bAdd THEN
	IF bNoAndTime THEN
		wMessageNo:=wMessageNo + 1;
		sMessage := CONCAT(CONCAT(CONCAT(CONCAT(CONCAT(WORD_TO_STRING(wMessageNo),'.$t'),sActTime),'$t'),sMessage),'$n');
	END_IF
	fbSaveEventBuffer.A_AddTail();
END_IF

CASE nStep OF
	0:
	(* Jesli jest komunikat do zapisania to zapisz *)
	IF fbSaveEventBuffer.nCount>0 THEN
		fbSaveEventBuffer.A_RemoveHead();
		fbSaveEvent.bExecute:=TRUE;
		nStep := nStep + 10;
	END_IF
	10:
	fbSaveEvent.bExecute:=FALSE;
	(* Jak zapis zakonczony sukcesem - to wroc do kroku 0 *)
	IF NOT bBusy AND NOT bError THEN
		nStep := 0;
	END_IF
	(* Jak blad to zresetuj bloczek i podejmij próbę ponownie *)
	IF bError THEN
		nStep := nStep + 10;
	END_IF
	20:
		fbSaveEvent.bExecute:=TRUE;
		nStep := nStep - 10;
END_CASE

fbSaveEvent(
	AmsNetId	:= AmsNetId,
	sPath		:= sPath,
	sName		:= sName,
	sLine		:= sFileMessage,
	bBusy		=> bBusy,
	bError		=> bError);

END_FUNCTION_BLOCK

// ---- POUs/FileAccess/FB_FilePutText.TcPOU
(****************************************************************************************)
(*							Beckhoff Automation Poland									*)
(*								FB_FilePutText  v1.0									*)
(*									26.06.2014											*)
(*				Blok funkcyjny pozwalający wpisać do pliku String(1000)					*)
(*						jest to rozszerzenie bloku FB_FilePuts							*)
(*______________________________________________________________________________________*)
FUNCTION_BLOCK FB_FilePutText			(* Write a string to a stream. *)
VAR_INPUT
	sNetId					:	T_AmsNetId;		(* ams net id *)
	hFile					:	UINT;			(* file handle *)
	sLine					:	STRING(1000);	(* string to write *)
	bExecute				:	BOOL;			(* control input *)
	tTimeout				:	TIME := DEFAULT_ADS_TIMEOUT;
END_VAR
VAR_OUTPUT
	bBusy					:	BOOL;
	bError					:	BOOL;
	nErrId					:	UDINT;
END_VAR
{library private}
VAR
	fbAdsRdWrt				:	FW_AdsRdWrt := ( nPort := AMSPORT_R3_SYSSERV, nIdxGrp := SYSTEMSERVICE_FPUTS, cbReadLen := 0, pReadBuff := 0 );
END_VAR

fbAdsRdWrt( sNetId := sNetId, nIdxOffs := hFile, cbWriteLen := SIZEOF(sLine)(*inclusive terminating NULL*), pWriteBuff := ADR(sLine),
			bExecute := bExecute, tTimeout := tTimeout, bBusy=>bBusy, bError=>bError, nErrID=>nErrID );

END_FUNCTION_BLOCK

// ---- POUs/FileAccess/FB_ReceipRW.TcPOU
(****************************************************************************************************)
(*							Beckhoff Automation Poland												*)
(*							FB_ReceipRW v1.1														*)
(*									17.09.2012														*)
(*		Blok funkcyjny zapisu i odczytu receptury (dowolnej zmiennej) w formie binarnej				*)
(*____________________________________________________________________________________________________
	Versions:
		v1.1	05.08.2016	* Przepisana wersja do TwinCat3
		v1.0	17.09.2012	* Podstawowa wersja z TwinCat2
____________________________________________________________________________________________________*)
FUNCTION_BLOCK FB_ReceipRW
VAR_INPUT
	sNetId			: T_AmsNetId;
	sPath			: STRING;
	sFileName		: STRING;
	bSave			: BOOL;
	pWriteBuff		: DWORD;
	cbWriteLen		: UDINT;
	bLoad			: BOOL;
	pReadBuff		: DWORD;
	cbReadLen		: UDINT;
END_VAR
VAR_OUTPUT
	bBusy			: BOOL;
	bError			: BOOL;
END_VAR
VAR
	rtSave			: R_TRIG;
	rtLoad			: R_TRIG;
	bSaveAction		: BOOL;
	bLoadAction		: BOOL;
	fbFileOpen		: FB_FileOpen;
	ftOpen			: F_TRIG;
	fbFileWrite		: FB_FileWrite;
	ftWrite			: F_TRIG;
	fbFileRead		: FB_FileRead;
	ftRead			: F_TRIG;
	fbFileClose		: FB_FileClose;
	ftClose			: F_TRIG;
	rtError			: R_TRIG;
END_VAR

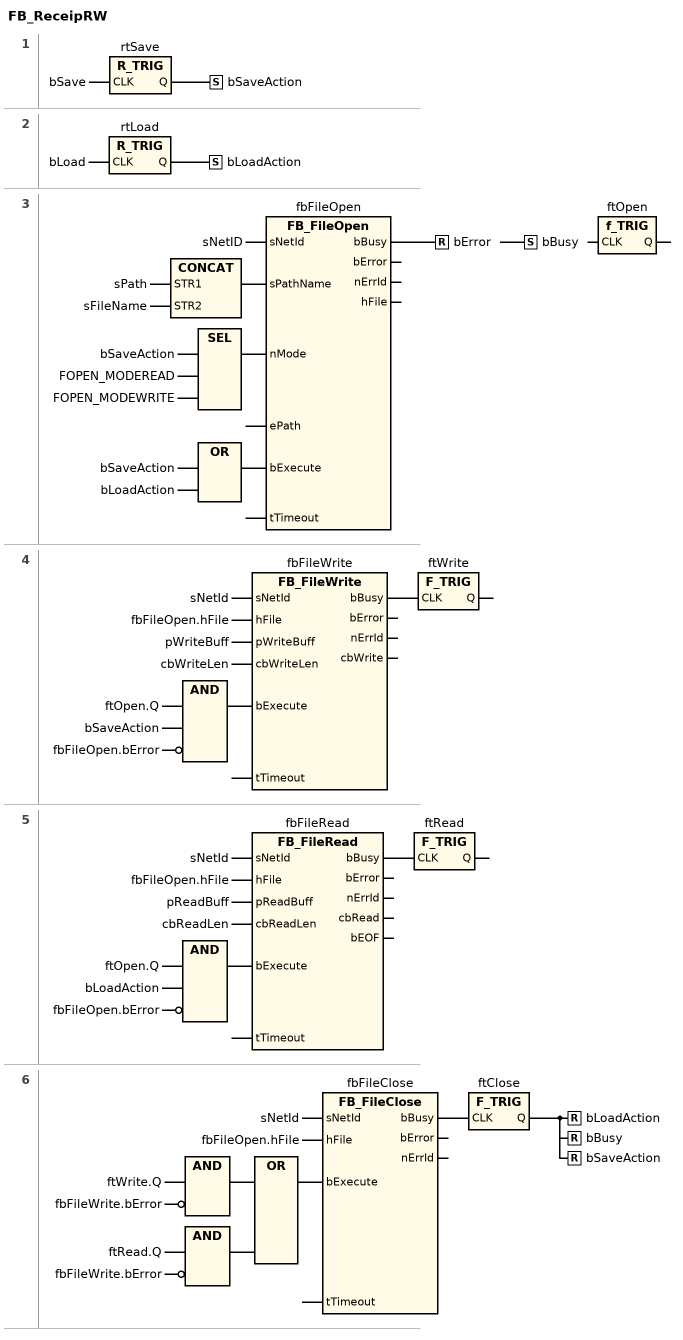
// NETWORK 1
rtSave(CLK := bSave); // R_TRIG
bSaveAction S= rtSave.Q;

// NETWORK 2
rtLoad(CLK := bLoad); // R_TRIG
bLoadAction S= rtLoad.Q;

// NETWORK 3
fbFileOpen(
    sNetId := sNetID,
    sPathName := CONCAT(STR1 := sPath, STR2 := sFileName),
    nMode := SEL(bSaveAction, FOPEN_MODEREAD, FOPEN_MODEWRITE),
    bExecute := bSaveAction OR bLoadAction); // FB_FileOpen
bError R= fbFileOpen.bBusy;
bBusy S= fbFileOpen.bBusy;
ftOpen(CLK := fbFileOpen.bBusy); // f_TRIG

// NETWORK 4
fbFileWrite(
    sNetId := sNetId,
    hFile := fbFileOpen.hFile,
    pWriteBuff := pWriteBuff,
    cbWriteLen := cbWriteLen,
    bExecute := ftOpen.Q AND bSaveAction AND NOT fbFileOpen.bError); // FB_FileWrite
ftWrite(CLK := fbFileWrite.bBusy); // F_TRIG

// NETWORK 5
fbFileRead(
    sNetId := sNetId,
    hFile := fbFileOpen.hFile,
    pReadBuff := pReadBuff,
    cbReadLen := cbReadLen,
    bExecute := ftOpen.Q AND bLoadAction AND NOT fbFileOpen.bError); // FB_FileRead
ftRead(CLK := fbFileRead.bBusy); // F_TRIG

// NETWORK 6
fbFileClose(
    sNetId := sNetId,
    hFile := fbFileOpen.hFile,
    bExecute := ftWrite.Q AND NOT fbFileWrite.bError OR ftRead.Q AND NOT fbFileWrite.bError); // FB_FileClose
ftClose(CLK := fbFileClose.bBusy); // F_TRIG
bLoadAction R= ftClose.Q;
bBusy R= ftClose.Q;
bSaveAction R= ftClose.Q;

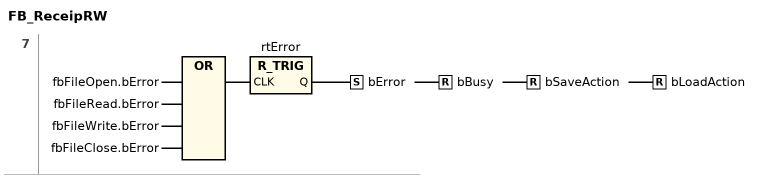
// NETWORK 7
rtError(CLK := fbFileOpen.bError OR fbFileRead.bError OR fbFileWrite.bError OR fbFileClose.bError); // R_TRIG
bError S= rtError.Q;
bBusy R= rtError.Q;
bSaveAction R= rtError.Q;
bLoadAction R= rtError.Q;

END_FUNCTION_BLOCK

// ---- POUs/FileAccess/FB_SaveLineToFile.TcPOU
(****************************************************************************************)
(*							Beckhoff Automation Poland									*)
(*								FB_SaveLineToFile  v2.0									*)
(*									26.06.2014											*)
(*						Blok funkcyjny zapisujacy tekst do pliku						*)
(*______________________________________________________________________________________
	Versions:
		v1.1	05.08.2016	* Przepisana wersja do TwinCat3
		v1.0	17.09.2012	* Podstawowa wersja z TwinCat2
________________________________________________________________________________________*)
FUNCTION_BLOCK FB_SaveLineToFile
VAR_INPUT
	bExecute	: BOOL;			(* Komenda wpisu *)
	AmsNetId	: T_AmsNetId;	(* AMS NET ID obiektu docelowego, gdy lokalnie, to zmienna moze byc pusta *)
	sPath		: STRING; 		(* Sciezka pliku, np  'Hard Disk\'*)
	sName		: STRING; 		(* Nazwa pliku wraz z rozszerzeniem 'LogFile.txt'; *)
	sLine		: STRING;		(* Tresc wpisu *)
END_VAR
VAR_OUTPUT
	bBusy		: BOOL;
	bError		: BOOL;
END_VAR
VAR
	fbFileOpen	: FB_FileOpen;
	ftOpen		: F_TRIG;
	fbFilePuts	: FB_FilePuts;
	ftPuts		: F_TRIG;
	fbFileClose	: FB_FileClose;
	ftClose		: F_TRIG;
END_VAR
VAR // added by the converter: edge detectors and wires of the graphical bodies
    _w1 : BOOL;
END_VAR

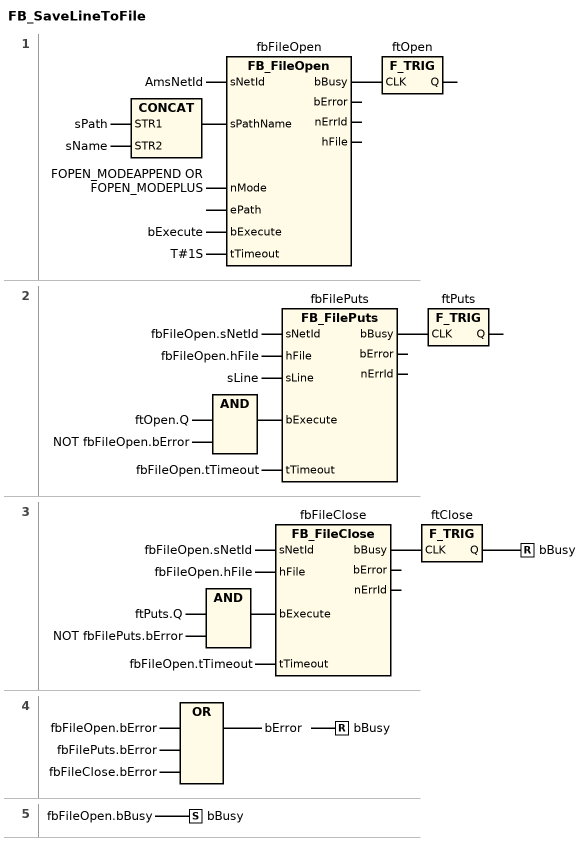
// NETWORK 1
fbFileOpen(
    sNetId := AmsNetId,
    sPathName := CONCAT(STR1 := sPath, STR2 := sName),
    nMode := FOPEN_MODEAPPEND OR FOPEN_MODEPLUS,
    bExecute := bExecute,
    tTimeout := T#1S); // FB_FileOpen
ftOpen(CLK := fbFileOpen.bBusy); // F_TRIG

// NETWORK 2
fbFilePuts(
    sNetId := fbFileOpen.sNetId,
    hFile := fbFileOpen.hFile,
    sLine := sLine,
    bExecute := ftOpen.Q AND (NOT fbFileOpen.bError),
    tTimeout := fbFileOpen.tTimeout); // FB_FilePuts
ftPuts(CLK := fbFilePuts.bBusy); // F_TRIG

// NETWORK 3
fbFileClose(
    sNetId := fbFileOpen.sNetId,
    hFile := fbFileOpen.hFile,
    bExecute := ftPuts.Q AND (NOT fbFilePuts.bError),
    tTimeout := fbFileOpen.tTimeout); // FB_FileClose
ftClose(CLK := fbFileClose.bBusy); // F_TRIG
bBusy R= ftClose.Q;

// NETWORK 4
_w1 := fbFileOpen.bError OR fbFilePuts.bError OR fbFileClose.bError;
bError := _w1;
bBusy R= _w1;

// NETWORK 5
bBusy S= fbFileOpen.bBusy;

END_FUNCTION_BLOCK

// ---- POUs/FileAccess/FB_WriteReportToFile.TcPOU
(****************************************************************************************************)
(*							Beckhoff Automation Poland												*)
(*							FB_WriteReportToFile v1.5												*)
(*					v1.2 - internal optimizations													*)
(*					v1.3 - internal optimizations													*)
(*					v1.4 - zmiana funkcjonalności, obsługa błędów, większa elastyczność				*)
(*					v1.5 - dodanie bufora zapisu, poprawienie zapisu Header							*)
(*									06.06.2012														*)
(*				Blok funkcyjny slużący do zapisywania danych do pliku *.xls.						*)
(*					Pierwszy wiersz kazdego pliku stanowi sHeader.									*)
(*	Zapisywane sData, podawane są na wejście bloku funkcyjnego jako zmienna typu STRING.			*)
(*				Pierwsza kolumna zawiera datę i godzinę wykonania wpisu.							*)
(*				Możliwe jest ustawienie częstości zapisywania do pliku,								*)
(* 			Konieczne jest dodanie biblioteki TcUtilities.lib, TcSystem.lib oraz TcBase.lib			*)
(*		UWAGA!!!																					*)
(*		Blok ten korzysta z czasu systemowego, podawanego na wejście bloku.							*)
(*		Nie można wywoływać tego bloku bez podania czasu na wejściu,								*)
(*		ponieważ wówczas przyjmuje on wartości zerowe i blok nie wykona zapisu						*)
(*		BLOK FUNKCYJNY DZIAŁA TYLKO DLA "PC OR CX( x86)"											*)
(*__________________________________________________________________________________________________*)

FUNCTION_BLOCK FB_WriteReportToFile
VAR_INPUT
	sHeader:				STRING(255);(*:='Czas$tKolumna1$tKolumna2$tKolumna3$n';*)(* Naglowki kolumn - cała górna linia - powinna być zakończona '$n'*)
 	sData: 					STRING(255);(*:='Zmienna1$tZmienna2$tZmienna3$n'; *)		(* sData do zapisu w postaci napisu, np 'test$n', 10 znaków zajmie stempel czasowy z przodu - dołączony zostanie automatycznie, więc max długość linii 245 znaków!!!!!! *)
	sPath:					STRING(255);(*:='c:\';*)										(* sPath zapisu pliku bez nazwy pliku, np 'c:\' *)
	stActTime:				TIMESTRUCT;												(* Aktualny czas w formie struktury - TIMESTRUCT*)
	tWriteFrequency:		TIME:=T#10s; 												(* Częstotliwość zapisu do pliku*)
	wNewFileFrequency:		WORD:=0;													(* Częstotliwość tworzenia nowego pliku: dzien (0), tydzien(1), miesiac(2) *)
	bWrite: 				BOOL; 														(* Zapis na rozkaz*)
END_VAR
VAR_OUTPUT
	bBusy: 					BOOL;		(* Sygnał zajętości bloczka *)
	bError:					BOOL;		(* Flaga błedu, bloczek sam się resetuje, więc flaga mnoże samoczynnie zniknąć *)
	dwErrors:				DWORD;	(* Suma błędów od uruchomienia programu PLC *)
	dwErrorsInCurrentFile:	DWORD;	(* Suma błedów zapisu do nowego pliku lub od uruchomienia *)
END_VAR

VAR
	sFileName: 				STRING;
	fbFileOpen: 			FB_FileOpen;
	fbFileWrite:  			FB_FilePuts;
	fbFileClose: 			FB_FileClose;
	Step: 					INT;
	TrigerName:				R_TRIG;
	sTime: 					STRING(10);(*odciecie min rozmiarem*)
	sTimeExcel: 			STRING(19);(*odciecie min rozmiarem*)
	stActTimeName:			TIMESTRUCT;												(* Aktualny czas w formie struktury użyty do tworzenia nazwy pliku *)
	sOldName:				STRING:='start';
	bInitialization: 		BOOL:=TRUE;
	WriteTimer: 			TON;
	WatchDog:				TON;
	rtWrite: 				R_TRIG; (* 1-krotny zapis na zadanie *)
	fbBuffer:				FB_StringRingBuffer;				(*Bufor zapisu*)
	arrBuffer: 				ARRAY [1..20] OF STRING(255);	(*Tablica bufora zapisu*)
	sLine:					STRING(255);						(*Linia do zapisu*)
END_VAR

(* Akcja wywołująca bloki w tle *)
CallBackgroundFBs();
(*Akcja Name*)
Name();
(*Obsługa bufora zapisu*)
fbBuffer(pBuffer:= ADR(arrBuffer),
		cbBuffer:= SIZEOF(arrBuffer));
(*Dodawanie elementów do bufora*)
IF rtWrite.Q OR WriteTimer.q  THEN
	fbBuffer.A_AddTail(putValue:= sData);
END_IF
CASE Step OF
	0: (* Initialization *)
		IF stActTime.wYear<>0 THEN
			(*format daty  w pliku Excela*)
			sTimeExcel:=SYSTEMTIME_TO_STRING(stActTime);
			WatchDog.IN:= TRUE;
			fbFileOpen.bExecute:= TRUE;
			bBusy := TRUE;
			bError := FALSE;
			bInitialization:=FALSE;
			fbFileOpen.bExecute := TRUE;
			fbFileOpen.nMode := FOPEN_MODEREAD;
			Step:= Step+5;
		END_IF
	5:	(*Sprawdzenie czy plik jest stworzony*)
		IF fbFileOpen.bBusy = FALSE AND NOT fbFileOpen.bError THEN
			Step := 60;
			sOldName := sFileName;
			fbFileOpen.bExecute := FALSE;
			fbFileClose.bExecute:= TRUE;
			fbFileOpen.nMode:= FOPEN_MODEAPPEND OR FOPEN_MODEPLUS ;
		ELSIF fbFileOpen.bError THEN
			Step := 20;
			fbFileOpen.bExecute := FALSE;
			fbFileOpen.nMode:= FOPEN_MODEAPPEND OR FOPEN_MODEPLUS ;
		END_IF
	10: (* Waiting for write request *)
		fbBuffer.A_RemoveHead(getValue=> sLine);
		IF fbBuffer.bOk AND sLine <> '' THEN
			(*format daty  w pliku Excela*)
			sTimeExcel:=SYSTEMTIME_TO_STRING(stActTime);
			WatchDog.IN:= TRUE;
			fbFileOpen.bExecute:= TRUE;
			bBusy := TRUE;
			bError := FALSE;
			Step := Step + 10;
		END_IF

	20:	(*Otwieramy plik*)
		fbFileOpen.bExecute := TRUE;
		IF fbFileOpen.bBusy = FALSE AND NOT fbFileOpen.bError THEN
			fbFileOpen.bExecute:= FALSE;
		(*Tworzene nowego pliku z naglowkiem*)
			IF sOldName = sFileName THEN
				(*do istniejacego pliku dopisujemy sData*)
				Step := Step + 20;
			ELSE
				(* Kasujemy błedy bieżącego pliku *)
				dwErrorsInCurrentFile := 0;
				(*Wysylamy sHeader*)
				fbFileWrite.bExecute:= TRUE;
				fbFileWrite.sLine := sHeader;
				sOldName := sFileName;
				Step := Step + 10;
			END_IF
		END_IF

	30:
		IF fbFileWrite.bBusy = FALSE AND NOT fbFileWrite.bError THEN
			fbFileWrite.bExecute:= FALSE;
			Step :=  50;
		END_IF

	40:	(*Wysylamy sLine*)
		fbFileWrite.bExecute:= TRUE;
		sTimeExcel := DELETE (sTimeExcel,1,11);(*usuniecie znaku' -' przed godzina*)
		sTimeExcel := INSERT (sTimeExcel,' ',10);(*wstawienie znaku ' ' przed godzina *)

		sLine:=CONCAT('$t',sLine);
		sLine:=CONCAT(sTimeExcel,sLine);
		fbFileWrite.sLine := sLine;
		Step := Step + 10;
	50:
		IF fbFileWrite.bBusy = FALSE AND NOT fbFileWrite.bError THEN
			fbFileWrite.bExecute:= FALSE;
			fbFileClose.bExecute:= TRUE;
			Step := Step + 10;
		END_IF

	60:	(*Zamykanie pliku*)
		IF fbFileClose.bBusy = FALSE AND fbFileClose.bError = FALSE THEN
			fbFileClose.bExecute:= FALSE;
			bBusy := FALSE;
			WatchDog.IN:= FALSE;
			Step := 10;
		END_IF
	99: (* Error *)
		fbFileOpen.bExecute:= FALSE;
		fbFileWrite.bExecute:= FALSE;
		fbFileClose.bExecute:= FALSE;
		WatchDog.IN:= FALSE;
		bError := TRUE;
		dwErrors := dwErrors + 1;
		dwErrorsInCurrentFile := dwErrorsInCurrentFile + 1;
		Step := 10;
END_CASE
CallFileFBs();

ACTION CallBackgroundFBs:
(*Wywolanie blokow funkcyjnych*)
TrigerName();
rtWrite(CLK:= bWrite);

(*Reset bloczka w przypadku bledu*)
WatchDog(PT:=T#10s);
IF WatchDog.Q THEN  Step:=99; END_IF

(*Ustalenie czestotliwosci zapisu do pliku*)
WriteTimer(IN:= NOT WriteTimer.Q, PT:= tWriteFrequency, Q=> , ET=> );
END_ACTION

ACTION CallFileFBs:
(*Wywołanie bloków odpowiedzialnych za zapisywanie*)
fbFileOpen(
	sNetId:= '',
	sPathName:= sFileName,
	ePath:= PATH_GENERIC,
	tTimeout:= T#200ms);

fbFileWrite(
	sNetId:= '',
	hFile:= fbFileOpen.hFile,
	tTimeout:= T#250ms);

fbFileClose(
	sNetId:= '',
	hFile:= fbFileOpen.hFile,
	tTimeout:= t#200ms);
END_ACTION

ACTION Name:
(*xxxxxxxxxxxxxxxxxxxxxxxxxxxxxxxxxxxxxxxxxxxxxxxxxxxxxxxxxxxxxxxxxxxxxxxxxxxxxxxxxxxxxxxxxxxxxxxxxxxxxxxxxxxxxxxx
				Ustalenie częstotliwości twrzenia nowego pliku i zmiana nazwy pliku
xxxxxxxxxxxxxxxxxxxxxxxxxxxxxxxxxxxxxxxxxxxxxxxxxxxxxxxxxxxxxxxxxxxxxxxxxxxxxxxxxxxxxxxxxxxxxxxxxxxxxxxxxxxxxxxxx*)
CASE wNewFileFrequency OF
	0:	(*Tworzenie pliku raz dziennie*)
		stActTimeName := stActTime;
		stActTimeName.wHour := 0;
		stActTimeName.wMinute := 0;

	1:	(*Tworzenie pliku raz w tygodniu*)
		IF bInitialization THEN
			stActTimeName := stActTime;
			stActTimeName.wHour := 0;
			stActTimeName.wMinute := 0;
		ELSIF stActTime.wDayOfWeek = 1 THEN
			stActTimeName := stActTime;
			stActTimeName.wHour := 0;
			stActTimeName.wMinute := 0;
		END_IF
ELSE
		(*Tworzenie pliku raz w miesiącu*)
		stActTimeName := stActTime;
		stActTimeName.wDay := 1;
		stActTimeName.wHour := 0;
		stActTimeName.wMinute := 0;

END_CASE

sTime := SYSTEMTIME_TO_STRING(stActTimeName);
sTime := DELETE (sTime,1,11);(*usuniecie znaku' -' przed godzina*)
sFileName:=CONCAT(sPath,sTime);
sFileName:=CONCAT(sFileName,'.xls');
END_ACTION

END_FUNCTION_BLOCK

// ---- POUs/FileAccess/FB_XCopyCE.TcPOU
(********************************************************************************************)
(*							Beckhoff Automation Poland										*)
(*								FB_XCopyCE  v1.0											*)
(*									07.07.2010												*)
(*	Bloczek kopiujący plik z miejsca zrodlowego do docelowego,  							*)
(*	jesli w miejscu docelowym jest juz plik o tej nazwie, zostanie on zastąpiony			*)
(*	BF wykorzystuje  NT_StartProcess znajudjący się w bibliotece TcUtilities.lib			*)
(*	Sprawdzony pod systemem Windows CE5 i CE6, wymaga pliku 	\Hard Disk\System\XCOPYCE	*)
(*__________________________________________________________________________________________*)
FUNCTION_BLOCK FB_XCopyCE
VAR_INPUT
	bCopy : 			BOOL;	(* zbocze narastajace rozpoczyna kopiowanie *)
	NetID: 				STRING;
	sFileName : 		STRING;	(* nazwa pliku np: 'a.txt' *)
	sSrcPath : 			STRING;	(* sciezka zrodlowa np: '\Hard Disk\' *)
	sDestPath :		 	STRING;	(* sciezka docelowa np: '\Hard Disk\ftp\' *)

END_VAR
VAR_OUTPUT
	bBusy : 			BOOL;
	bError :	 		BOOL;
	bErrID :			UDINT;
END_VAR
VAR
	NtStartProcess : 	NT_StartProcess;
	rtCopy: 			R_TRIG;
	step: 				INT;
	sCmd: 				STRING;
END_VAR

rtCopy(CLK:= bCopy, Q=> );

IF rtCopy.Q THEN 	step := step +10; END_IF

CASE step OF
0:	(* czeka na polecenie kopiowania *)
	bBusy:= FALSE;
	NtStartProcess.START := FALSE;
10:
	bBusy := TRUE;
	bError := FALSE;
	bErrID :=0;
	sCmd:='';				(* tworzenie polecenia *)
	sCmd := CONCAT(CONCAT(CONCAT('"', sSrcPath), sFileName), '" "');
	sCmd := CONCAT(CONCAT(sCmd, sDestPath), '" /Y');
	NtStartProcess.START := TRUE;
	step := step +10;

20:
	IF NOT NtStartProcess.BUSY AND NOT NtStartProcess.ERR THEN
		step := Step -20;
	ELSIF  NtStartProcess.ERR THEN
		Step := step -20;
		bError := TRUE;
		bErrID := NtStartProcess.ERRID;
	END_IF
END_CASE



NtStartProcess(
	NETID:= NetID,
	PATHSTR:=  '\Hard Disk\System\XCOPYCE',
	DIRNAME:=  '\Hard Disk\System',
	COMNDLINE:= sCmd ,
	START:= ,
	TMOUT:= ,
	BUSY=> ,
	ERR=> , 
	ERRID=> );

END_FUNCTION_BLOCK

// ---- POUs/FlipFlop/FB_toggle.TcPOU
(****************************************************************************************)
(*							Beckhoff Automation Poland									*)
(*								FB_Toogle  v1											*)
(*									27.05.2008											*)
(*				Bloczek do zamiany wartosci out z 1 na 0 i z 0 na 1						*)
(*______________________________________________________________________________________*)

FUNCTION_BLOCK FB_toggle
VAR_INPUT
	bIn:		BOOL;(*wartosc wejsciowa*)
END_VAR
VAR_OUTPUT
	bOut:		BOOL;(*wartosc wyjsciowa*)
END_VAR
VAR
	lastin:		BOOL:=TRUE;
	lastout:	BOOL;
END_VAR

bOut:=SEL(bIn>lastin,bOut,NOT bOut);
lastout:=bOut;
lastin:=bIn;

END_FUNCTION_BLOCK

// ---- POUs/FlipFlop/FB_TOGGLE_WITH_RESET.TcPOU
(********************************************************************************************)
(*							Beckhoff Automation Poland										*)
(*								FB_XCopyCE  v1.0											*)
(*									07.07.2010												*)
(*	Bloczek kopiujący plik z miejsca zrodlowego do docelowego,  							*)
(*	jesli w miejscu docelowym jest juz plik o tej nazwie, zostanie on zastąpiony			*)
(*	BF wykorzystuje  NT_StartProcess znajudjący się w bibliotece TcUtilities.lib			*)
(*	Sprawdzony pod systemem Windows CE5 i CE6, wymaga pliku 	\Hard Disk\System\XCOPYCE	*)
(*__________________________________________________________________________________________*)
FUNCTION_BLOCK FB_TOGGLE_WITH_RESET
VAR_INPUT
	bCopy : 			BOOL;	(* zbocze narastajace rozpoczyna kopiowanie *)
	NetID: 				STRING;
	sFileName : 		STRING;	(* nazwa pliku np: 'a.txt' *)
	sSrcPath : 			STRING;	(* sciezka zrodlowa np: '\Hard Disk\' *)
	sDestPath : 		STRING;	(* sciezka docelowa np: '\Hard Disk\ftp\' *)

END_VAR
VAR_OUTPUT
	bBusy : 			BOOL;
	bError : 			BOOL;
	bErrID :			UDINT;
END_VAR
VAR
	NtStartProcess: 	NT_StartProcess;
	rtCopy: 			R_TRIG;
	step: 				INT;
	sCmd: 				STRING;
END_VAR

rtCopy(CLK:= bCopy, Q=> );

IF rtCopy.Q THEN 	step := step +10; END_IF

CASE step OF
0:	(* czeka na polecenie kopiowania *)
	bBusy:= FALSE;
	NtStartProcess.START := FALSE;
10:
	bBusy := TRUE;
	bError := FALSE;
	bErrID :=0;
	sCmd:='';				(* tworzenie polecenia *)
	sCmd := CONCAT(CONCAT(CONCAT('"', sSrcPath), sFileName), '" "');
	sCmd := CONCAT(CONCAT(sCmd, sDestPath), '" /Y');
	NtStartProcess.START := TRUE;
	step := step +10;

20:
	IF NOT NtStartProcess.BUSY AND NOT NtStartProcess.ERR THEN
		step := Step -20;
	ELSIF  NtStartProcess.ERR THEN
		Step := step -20;
		bError := TRUE;
		bErrID := NtStartProcess.ERRID;
	END_IF
END_CASE



NtStartProcess(
	NETID:= NetID,
	PATHSTR:=  '\Hard Disk\System\XCOPYCE',
	DIRNAME:=  '\Hard Disk\System',
	COMNDLINE:= sCmd ,
	START:= ,
	TMOUT:= ,
	BUSY=> ,
	ERR=> , 
	ERRID=> );

END_FUNCTION_BLOCK

// ---- POUs/FlipFlop/FB_TypeJK.TcPOU
(************************************************************************************************************)
(*							Beckhoff Automation Poland														*)
(*								FB_TypeJK  v1																*)
(*									27.05.2008																*)
(*	Bloczek przerzutnika JK																					*)
(*	Przerzutnik ma wejścia informacyjne (J i K), , wyjście proste (Q) i jego negację (nie Q),				*)
(*	Przerzutnik jest przerzutnikiem synchronicznym, co oznacza, że zmienia stan przy zmianie stanu wejścia 	*)
(*	zegarowego z niskiego na wysoki (0 na 1)-wyzwalanie zboczem narastającym lub przy zmianie stanu			*)
(*	wejścia zegarowego(CLK) z wysokiego na niski (1 na 0)- wyzwalanie zboczem opadającym .					*)
(*	Stan wyjść podczas pracy przerzutnika zależy od stanu wejść, jak i stanu poprzedniego wyjść.			*)
(*__________________________________________________________________________________________________________*)
FUNCTION_BLOCK FB_TypeJK
VAR_INPUT
	J:			BOOL;
	Clk:		BOOL;
	K:			BOOL;
END_VAR
VAR_OUTPUT
	Q:			BOOL;
END_VAR
VAR
	lastClk:	BOOL;
	lastQ: 		BOOL;
END_VAR

IF (lastClk < Clk) THEN
	IF(J=1 AND K=0) THEN Q:=0; END_IF
	IF(J=0 AND K=1) THEN Q:=1; END_IF
	IF(J=1 AND K=1) THEN Q:=NOT lastQ; END_IF
	IF(J=0 AND K=0) THEN Q:=lastQ; END_IF
END_IF
lastQ:=Q;
lastClk:=Clk;

END_FUNCTION_BLOCK

// ---- POUs/FlipFlop/FB_TypeJK_SEL.TcPOU
(************************************************************************************************************)
(*							Beckhoff Automation Poland														*)
(*								FB_TypeJK_Sel  v1															*)
(*									27.05.2008																*)
(*	Bloczek przerzutnika JK z uzyciem funckji SEL(select)													*)
(*	Przerzutnik ma wejścia informacyjne (J i K), , wyjście proste (Q) i jego negację (nie Q),				*)
(*	Przerzutnik jest przerzutnikiem synchronicznym, co oznacza, że zmienia stan przy zmianie stanu wejścia 	*)
(*	zegarowego z niskiego na wysoki (0 na 1)-wyzwalanie zboczem narastającym lub przy zmianie stanu			*)
(*	wejścia zegarowego(CLK) z wysokiego na niski (1 na 0)- wyzwalanie zboczem opadającym .					*)
(*	Stan wyjść podczas pracy przerzutnika zależy od stanu wejść, jak i stanu poprzedniego wyjść.			*)
(*__________________________________________________________________________________________________________*)
FUNCTION_BLOCK FB_TypeJK_SEL
VAR_INPUT
	J:			BOOL;
	Clk:		BOOL;
	K:			BOOL;
END_VAR
VAR_OUTPUT
	Q:			BOOL;
END_VAR
VAR
	lastClk:	BOOL;
	lastQ: 		BOOL;
END_VAR

IF (lastClk<Clk) THEN
	Q:=SEL(J=1 AND K=0,Q,FALSE);
	Q:=SEL(J=0 AND K=1,Q,TRUE);
	Q:=SEL(J=1 AND K=1,Q,NOT lastQ);
	Q:=SEL(J=0 AND K=0,Q,lastQ);
END_IF
lastQ:=Q;
lastClk:=Clk;

END_FUNCTION_BLOCK

// ---- POUs/FlipFlop/FB_TypeRS.TcPOU
(****************************************************************************************************)
(*							Beckhoff Automation Poland												*)
(*								FB_TypeRS  v1														*)
(*									27.05.2008														*)
(*	Bloczek porzerzutnika typu RS																	*)
(*	Jeśli na wejściu zegarowym jest stan nieaktywny to przerzutnik nie reaguje na zmiany			*)
(*	sygnałów na pozostałych wejściach. Jeśli natomiast na wejściu zegarowym jest stan aktywny 		*)
(*	przerzutnik zmienia się zgodnie z tablicą (dla przerzutnika typu RS)	.						*)
(*	Różnie można rozumieć stan aktywny oraz stan nieaktywny - jest to zależne od wykonania			*)
(*	przerzutnika. Może to być:																		*)
(*    * Stan niski - 0 (Wyzwalanie niskim poziomem sygnału zegarowego)								*)
(*   * Stan wysoki - 1 (Wyzwalanie wysokim poziomem sygnału zegarowego)								*)
(*    * Moment zmiany stanu z niskiego na wysoki (0 na 1)											*)
 (*   * Moment zmiany stanu z wysokiego na niski (1 na 0) 											*)
(*__________________________________________________________________________________________________*)
FUNCTION_BLOCK FB_TypeRS
VAR_INPUT
	bR:			BOOL;
	bS:			BOOL;
END_VAR
VAR_OUTPUT
	bQ:			BOOL;
END_VAR
VAR
END_VAR

IF(bR =1) THEN bQ:=0;
ELSIF(bS=1) THEN bQ:=1;
END_IF

END_FUNCTION_BLOCK

// ---- POUs/FlipFlop/FB_TypeSR.TcPOU
(****************************************************************************************)
(*							Beckhoff Automation Poland									*)
(*								FB_TypeSR  v1											*)
(*									27.05.2008											*)
(*				Bloczek przerzutnika SR	(przewaga SET)									*)
(*______________________________________________________________________________________*)
FUNCTION_BLOCK FB_TypeSR
VAR_INPUT
	bR:			BOOL;
	bS:			BOOL;
END_VAR
VAR_OUTPUT
	bQ:			BOOL;
END_VAR
VAR
END_VAR

IF(bS=1) THEN bQ:=1;
ELSIF(bR=1) THEN bQ:=0;
END_IF

END_FUNCTION_BLOCK

// ---- POUs/HVAC/FB_AirMixer.TcPOU
(****************************************************************************************)
(*							Beckhoff Automation Poland									*)
(*								FB_AiRMixer  v1											*)
(*									27.05.2008											*)
(*							Bloczek do mieszania powietrza								*)
(*______________________________________________________________________________________*)
FUNCTION_BLOCK FB_AirMixer
VAR_INPUT
	Set:			REAL;
	Tin:			REAL;
	Tout:			REAL:=1;
	UpperLimit:		REAL;
	LowerLimit:		REAL;
END_VAR
VAR_OUTPUT
	Y:				REAL;
	Cool:			BOOL;
	Heat:			BOOL;
END_VAR
VAR
	deltaT:			REAL;
	a:				REAL;
	b:				REAL;
	Wyjscie: 		REAL;
	deltaLimit: 	REAL;
END_VAR

deltaT:=Tout-Tin;
deltaLimit:=UpperLimit-LowerLimit;
(*a:=deltaLimit/deltaT;*)
(*b:=(-deltaLimit*Tin)/deltaT;*)
Wyjscie:=a*Set+b;
IF Wyjscie < LowerLimit THEN
	Y:= LowerLimit;
	Cool:=TRUE;
ELSE Y:=Wyjscie;
END_IF
IF Wyjscie >UpperLimit THEN
	 Y:= UpperLimit;
	Heat:=TRUE;
ELSE Y:= Wyjscie;
END_IF
IF cool = TRUE AND Wyjscie>(LowerLimit+0.2*deltaLimit) THEN cool:=FALSE; END_IF
IF heat = TRUE AND Wyjscie>(UpperLimit-0.2*deltaLimit) THEN heat:=FALSE; END_IF

END_FUNCTION_BLOCK

// ---- POUs/HVAC/FB_Alarm.TcPOU
(********************************************************************************************)
(*							Beckhoff Automation Poland										*)
(*								FB_Alarm  v1												*)
(*									27.05.2008												*)
(*				Podstawowy blok funkcyjny kontroli alarmow									*)
(*__________________________________________________________________________________________*)
FUNCTION_BLOCK FB_Alarm
VAR_INPUT
	bIn:		BOOL;	(*sygnal wejsciowy alarmu*)
	bAck:		BOOL;	(*sygnal potwierdzenia alarmu*)
END_VAR
VAR_OUTPUT
	bOut1:		BOOL;	(*gdy zmienna =1  wystapil alarm*)
	bOut2:		BOOL;	(*gdy zmienna = 1 wystapil alarm  i nie zostal zatwierdzony*)
END_VAR
VAR
	lastin: 	BOOL;
	lastAck: 	BOOL;
END_VAR

IF lastIn<bIn THEN bOut1:=TRUE; bOut2:=TRUE; END_IF(*wystapil alarm*)
IF lastAck<bAck AND bIn THEN bOut1:=TRUE; bOut2:=FALSE; END_IF(*alarm zostal zatwierdzony ale wciaz wystepuje  *)
IF lastAck<bAck AND NOT bIn THEN bOut1:=FALSE; bOut2:=FALSE; END_IF
IF lastIn>bIn AND bOut2=FALSE THEN bOut1:=FALSE; END_IF
lastIn:=bIn;
lastAck:=bAck;

END_FUNCTION_BLOCK

// ---- POUs/HVAC/FB_Boiler_Load.TcPOU
(****************************************************************************************)
(*							Beckhoff Automation Poland									*)
(*								FB_Boiler_Load  v1										*)
(*									27.05.2008											*)
(*						Bloczek do kontroli grzania boilera								*)
(*______________________________________________________________________________________*)
FUNCTION_BLOCK FB_Boiler_Load
VAR_INPUT
	TempUp:			INT;(**)
	TempDown:		INT;(**)
	Enable:			BOOL;(*wlaczenie*)
	Off:			INT;(**)
	On:				INT;(**)
END_VAR
VAR_OUTPUT
	Out: 			BOOL:= FALSE;
END_VAR

IF Enable THEN
	IF TempUp < On THEN Out := TRUE; END_IF(*gdy temp zadana wyzsza od temp aktualnej wlacza boiler*)
	IF Tempdown > Off THEN Out := FALSE; END_IF
END_IF

END_FUNCTION_BLOCK

// ---- POUs/HVAC/FB_Controller2Point.TcPOU
(****************************************************************************************)
(*							Beckhoff Automation Poland									*)
(*								FB_Controller2Point  v1									*)
(*									06.10.2016											*)
(*	Bloczek do regulatora 2 stawnego													*)
(*	MinLimit < MaxLimit																	*)
(*______________________________________________________________________________________*)
FUNCTION_BLOCK FB_Controller2Point
VAR_INPUT
	rIn			:	REAL;(*wartosc wejsciowa*)
	rMinLimit	:	REAL;(*wartosc dolna regulatora*)
	rMaxLimit	:	REAL;(*wartosc gorna regulatora*)
END_VAR
VAR_OUTPUT
	bOut		:	BOOL;(*wyjscie regulatora*)
END_VAR

bOut:=SEL(rIn<rMinLimit,bOut,TRUE);(*gdy wartosc zadana jest mniejsza od wartosci mniejszej zalacza wyjscie*)
bOut:=SEL(rIn>rMaxLimit,bOut,FALSE);(*gdy wartosc zadana jest wieksza od wartosci maksymalnej wylacza wyjscie*)

END_FUNCTION_BLOCK

// ---- POUs/HVAC/FB_DeadNullRange.TcPOU
(****************************************************************************************)
(*							Beckhoff Automation Poland									*)
(*								FB_DeadNullRange  v1									*)
(*									27.05.2008											*)
(*					Bloczek do kontroli strefy nieczulosci								*)
(*______________________________________________________________________________________*)
FUNCTION_BLOCK FB_DeadNullRange
VAR_INPUT
	In:			REAL;(*sygnal wejsciowy*)
	Dead:		REAL;(**)
	Null:		REAL;(**)
END_VAR
VAR_OUTPUT
	Out:		REAL;(*sygnal wyjsciowy*)
END_VAR

IF(In<Null AND In>-Null) THEN Out:=0;
ELSE
	IF(In>Out+Dead OR In< Out-Dead) THEN Out:=In;	END_IF
END_IF

END_FUNCTION_BLOCK

// ---- POUs/HVAC/FB_LimitHVAC.TcPOU
(************************************************************************************************)
(*							Beckhoff Automation Poland											*)
(*								FB_LimitHVAC  v1												*)
(*									27.05.2008													*)
(*	Bloczek do kontroli temperatury z zadanymi wartosciami minimalna i maksymalna				*)
(*	gdy temp jest z  przedzialu (MiniOut,MaxOut) to na wyjsciu pojawia sie temp z wejscia		*)
(*	w przeciwnym razie pokazuje sie ostatania wskazywana temperatura							*)
(*______________________________________________________________________________________________*)
FUNCTION_BLOCK FB_LimitHVAC
VAR_INPUT
	In:			REAL;
	MaxOut:		REAL;
	MiniOut:	REAL;
END_VAR
VAR_OUTPUT
	Out:		REAL;
END_VAR

Out:= SEL(In>MaxOut,Out,MaxOut);
Out:= SEL(In<MiniOut,Out,MiniOut);
Out:= SEL(In>MiniOut AND In<MaxOut,Out,In);

END_FUNCTION_BLOCK

// ---- POUs/HVAC/FB_SeqCMH.TcPOU
(****************************************************************************************************)
(*							Beckhoff Automation Poland												*)
(*								FB_SeqCMH  v1														*)
(*									27.05.2008														*)
(*	Bloczek do kontroli  ogrzewania,chlodzenia														*)
(*	jezeli temp(X) jest wieksza od zadanych wartosci podanych w przedzialach to wykonywane sa 		*)
(*	dzialania majace na celu podanie na wyjsciu wartosciu w procent. Trzeba podac na wejsciu		*)
(*	ktora wartosc chce sie otrzymac poprzez podanie na wejsciach : enC,enM;enH	wartosci 1			*)
(*																									*)
(*__________________________________________________________________________________________________*)
FUNCTION_BLOCK FB_SeqCMH
VAR_INPUT
	X:				REAL;(*sygnal wejsciowy*)
	enC:			BOOL;(*zmienna odpowiedzialna za uruchomienie chlodzenia Cooling*)
	enM:			BOOL;(*zmienna odpowiedzialna za uruchomienie chlodzenia Mixing*)
	enH:			BOOL;(*zmienna odpowiedzialna za uruchomienie grzania Heating*)
	CoolingLow:		REAL;(*zmienna z zakresu dolnego do chlodzenia*)
	CoolingHi:		REAL;(*zmienna z zakresu gornego do chlodzenia*)
	MLow:			REAL;(*zmienna z zakresu dolnego*)
	MHi:			REAL;(*zmienna z zakresu gornego*)
	HeatLow:		REAL;(*zmienna z zakresu dolnego do ogrzewania*)
	HeatHi:			REAL;(*zmienna z zakresu gornego do ogrzewania*)
	Tinside:		REAL;(**)
	Toutside:		REAL;(**)
END_VAR
VAR_OUTPUT
	OutC:			REAL;(*zmienna wyjsciowa chlodzenia*)
	OutM:			REAL;(**)
	OutH:			REAL;(*zmienna wyjsciowa ogrzewania*)
END_VAR
VAR
END_VAR

IF X>=CoolingLow AND X<=CoolingHi AND enC THEN
	OutC:= (CoolingHi-X)*100/(CoolingHi-CoolingLow);
	OutM:=0;
	OutH:=0;
END_IF
IF X>=MLow AND X<=MHi AND enM  THEN
	IF Tinside > Toutside THEN
		OutC:=0;
		OutM:= (MHi-X)*100/(MHi-MLow);
		OutH:=0;
	ELSE
		OutC:=0;
		OutM:= 100- (MHi-X)*100/(MHi-MLow);
		OutH:=0;
	END_IF
END_IF

IF X>=HeatLow AND X<=HeatHi AND enH THEN
	OutC:=0;
	OutM:=0;
	OutH:= (X-HeatLow)*100/(HeatHi-HeatLow);
END_IF

IF NOT enC THEN outC:=0; END_IF
IF NOT enM THEN outM:=0; END_IF
IF NOT enH THEN outH:=0; END_IF

END_FUNCTION_BLOCK

// ---- POUs/KL_Terminals/FB_KL320x_1channel.TcPOU
(****************************************************************************************)
(*							Beckhoff Automation Poland									*)
(*							FB_KL320x_1channel v1.1										*)
(*									9.11.2007											*)
(*		Blok funkcyjny konfigurujący kanał modułu KL320x dla określonego typu czujnika	*)
(*							Współpracuje z modułem KL320x.								*)
(*______________________________________________________________________________________*)

FUNCTION_BLOCK FB_KL320x_1channel
(*Objaśnienie procedur*)
(*	Control Byte
	BIT7 = 1 Register Mode
	BIT6 = 0 Read Register
	BIT6 = 1 Write Register
	BIT5-BIT0 -> Register Number
	
	usStatus BYTE
	BIT7 -> Writing Acknowledgement
	BIT5-BIT0 -> Which Register was Read
	
	R31 - CodeWord Register Code: 16#1235

	R32 - Feature Register:
					BIT15	BIT14	BIT13	BIT12	Element		Measuring Range
usSensorType = 0		0		0		0		0		PT100		-200C 	+850C
usSensorType = 1		0		0		0		1		NI100		-60C 	+250C
usSensorType = 2		0		0		1		0		PT1000		-200C	+850C
usSensorType = 3		0		0		1		1		PT500		-200C	+850C
usSensorType = 4		0		1		0		0		PT200		-200C	+850C
usSensorType = 5		0		1		0		1		NI1000		-200C	+850C
usSensorType = 6		0		1		1		0		NI120		-200C	+850C
usSensorType = 7		1		1		1		0		Output in Ohm	10.0		5000.0 Ohm
usSensorType = 8 	1		1		1		1		Output in Ohm 10.0		1200.0 Ohm
*)
VAR_INPUT
	bChange:			BOOL;		(*Rising edge activated function block*)
	usSensorType:		USINT;		(*Sensor type*)
	usState :			USINT;		(*Linked with KL320x - Channel X - Status*)
	iDataIn:			INT;		(*Linked with KL320x - Channel X - DataIn*)
END_VAR
VAR_OUTPUT
	bDone:				BOOL;		(*If the execution of the function block is without error this output is set*)
	bError:				BOOL;		(*If an error is occur during the execution of the function block this output is set*)
	usCtrl:				USINT;		(*Linked with KL320x - Channel X - Ctrl*)
	iDataOut:			INT;		(*Linked with KL320x - Channel X - DataOut*)
END_VAR
VAR
	Step: 				USINT;
	Trig1:				R_TRIG;
END_VAR
VAR CONSTANT
	CodeWordRegister: 	BYTE := 31;
	FeatureRegister: 	BYTE := 32;
	Code: 				WORD := 16#1235;
END_VAR

Trig1(CLK:= bChange);
IF Trig1.Q  THEN
	Step := 1;
END_IF
CASE Step OF
	0:
		usCtrl := 0;
		iDataOut := 0;

	1:	(*Write Code*)
		usCtrl := CodeWordRegister;
		usCtrl.7 := TRUE;(*tryb register comm*)
		usCtrl.6 := TRUE;(*true -zaspis rejestru, false - odczyt*)
		iDataOut := word_to_int(Code);
		Step := Step + 1;

	2:	Step := Step + 1;(*czekamy*)

	3:	(*Read if Code write was succesful*)
		IF usCtrl.7 THEN
			Step := Step + 1;
		ELSE
			bError := TRUE;
			Step := 0;
		END_IF

	4:	(*Read Feature Register*)
		usCtrl := FeatureRegister;
		usCtrl.7 := TRUE;
		usCtrl.6 := FALSE;
		Step := Step + 1;

	5:	Step := Step + 1;

	6:
		usCtrl := FeatureRegister;
		usCtrl.7 := TRUE;
		usCtrl.6 := TRUE;
		iDataOut := iDataIn;(*Leave other settings*)
		CASE usSensorType OF
			0:	iDataOut.15 := FALSE;	iDataOut.14 := FALSE;	iDataOut.13 :=	FALSE;	iDataOut.12 := FALSE;(*PT100*)
			1:	iDataOut.15 := FALSE;	iDataOut.14 := FALSE;	iDataOut.13 :=	FALSE;	iDataOut.12 := TRUE;(*NI100*)
			2:	iDataOut.15 := FALSE;	iDataOut.14 := FALSE;	iDataOut.13 :=	TRUE;	iDataOut.12 := FALSE;(*PT1000*)
			3:	iDataOut.15 := FALSE;	iDataOut.14 := FALSE;	iDataOut.13 :=	TRUE;	iDataOut.12 := TRUE;(*PT500*)
			4:	iDataOut.15 := FALSE;	iDataOut.14 := TRUE;	iDataOut.13 :=	FALSE;	iDataOut.12 := FALSE;(*PT200*)
			5:	iDataOut.15 := FALSE;	iDataOut.14 := TRUE;	iDataOut.13 :=	FALSE;	iDataOut.12 := TRUE;(*NI1000*)
			6:	iDataOut.15 := FALSE;	iDataOut.14 := TRUE;	iDataOut.13 :=	TRUE;	iDataOut.12 := FALSE;(*NI120*)
			7:	iDataOut.15 := TRUE;	iDataOut.14 := TRUE;	iDataOut.13 :=	TRUE;	iDataOut.12 := FALSE;(*Output in Ohm 10.0 to 5000.0*)
			8:	iDataOut.15 := TRUE;	iDataOut.14 := TRUE;	iDataOut.13 :=	TRUE;	iDataOut.12 := TRUE;(*Output in Ohm 10.0 to 1200.0*)
		ELSE
			;
		END_CASE
		Step := Step + 1;

	7:	Step := Step + 1;(*Czekamy*)

	8:	IF usState.7  THEN
			bDone := TRUE;
			bError := FALSE;
		ELSE
			bDone := FALSE;
			bError := TRUE;
		END_IF
		Step := 100;

	100:	(*Write 0 to CodeWord Register back*)
		usCtrl	:= CodeWordRegister;
		usCtrl.7 := TRUE;
		usCtrl.6 := TRUE;
		iDataOut := 0;
		Step :=0;
END_CASE

END_FUNCTION_BLOCK

// ---- POUs/KL_Terminals/FB_KL32x8_1channel.TcPOU
(****************************************************************************************************)
(*							Beckhoff Automation Poland												*)
(*							FB_KL32x8_1channel v1.1													*)
(*									7.07.2015														*)
(* 				v1.1 - dodano wpis do rejestru R39 oraz wyjscie bBusy.								*)
(*				Zmiana nazw zmiennych zgodnie z notacja węgierska									*)
(*		Blok funkcyjny konfigurujący kanał modułu KL32x8 dla określonego typu czujnika				*)
(*__________________________________________________________________________________________________*)

FUNCTION_BLOCK FB_KL32x8_1channel
(*Objaśnienie procedur*)
(*	Control Byte
	BIT7 = 1 Register Mode
	BIT6 = 0 Read Register
	BIT6 = 1 Write Register
	BIT5-BIT0 -> Register Number
	
	usStatus BYTE
	BIT7 -> Writing Acknowledgement
	BIT5-BIT0 -> Which Register was Read
	
	R31 - CodeWord Register Code: 16#1235*)
VAR_INPUT
	bChange:				BOOL;	(*Rising edge activated function block*)
	bySensorType:			BYTE;	(*Sensor type	R32 - Feature Register:
													BIT15	BIT14	BIT13	BIT12	Element	
								bySensorType = 0		0		0		0		0		PT1000
								bySensorType = 1		0		0		0		1		NI1000
								bySensorType = 2		0		0		1		0		RSNI1000*)
	byFurtherElements: 		BYTE; (* R39: Further elements (supported by KL3208-0010, from firmware version 1C and hardware version 01)
									  50 	NCT1K8			-40°C ... 130°C
									  51 	NCT1K8_TK		-30°C ... 150°C
									  52 	NCT2K2			-50°C ... 130°C
									  53 	NCT3K			-50°C ...   80°C
									  54 	NCT5K			-40°C ... 100°C
									  55 	NTC10K			-30°C ... 150°C
									  56 	NTC10KPRE		-30°C ... 150°C
									  57 	NTC10K_3204	-40°C ... 110°C
									  58 	NTC10KTYP2	-50°C ... 130°C
									  59 	NTC10KTYP3	-50°C ... 130°C
									  60 	NTC10KDALE	-50°C ... 130°C
									  61 	NTC10K3A221	-40°C ... 130°C
									  62 	NTC20K			-20°C ... 150°C
									100		Poti, resolution 0.1 Ohm	0 ... 5 kOhm
									101 	Poti, resolution 1 Ohm	0 ... 10 kOhm
									200 	NTC100K		-40°C ... 130°C
									255 	user defined NTC*)
	usiState :				USINT;	(*Linked with KL32x8 - Channel X - Status*)
	iDataIn:				INT;	(*Linked with KL32x8 - Channel X - DataIn*)
END_VAR
VAR_OUTPUT
	bBusy: 					BOOL; 	(* FB has job *)
	bDone:					BOOL;	(*If the execution of the function block is without error this output is set*)
	bError:					BOOL;	(*If an error is occur during the execution of the function block this output is set*)
	usiCtrl:				USINT;	(*Linked with KL32x8 - Channel X - Ctrl*)
	iDataOut:				INT;	(*Linked with KL32x8 - Channel X - DataOut*)
END_VAR
VAR
	byStep: 				BYTE;
	rtChange:				R_TRIG;
END_VAR
VAR CONSTANT
	byCodeWordReg: 			BYTE := 31;
	byFeatureReg: 			BYTE := 32;
	byFurtherElementsReg: 	BYTE := 39;
	wCodeWord:				WORD := 16#1235;
END_VAR

rtChange(CLK:= bChange);
IF rtChange.Q  THEN
	byStep := 10;
	bBusy := TRUE;
	bDone := FALSE;
	bError := FALSE;
END_IF
CASE byStep OF
	0:
		usiCtrl := 0;
		iDataOut := 0;

	10:	(*Write Code*)
		usiCtrl := byCodeWordReg;
		usiCtrl.7 := TRUE;(*tryb register comm*)
		usiCtrl.6 := TRUE;(*true -zaspis rejestru, false - odczyt*)
		iDataOut := word_to_int(wCodeWord);
		byStep := byStep + 10;

	20:	byStep := byStep + 10;(*czekamy*)

	30:	(*Read if Code write was succesful R31 Read*)
		IF usiState = 2#1001_1111 THEN
			(*Read Feature Register*)
			usiCtrl := byFeatureReg;
			usiCtrl.7 := TRUE;
			usiCtrl.6 := FALSE;
		ELSE
			bBusy := FALSE;
			bError := TRUE;
		END_IF
		(* Jak nie ma bledy to dalej, jak blad to do kroku bledu *)
		IF bError THEN byStep := 255; ELSE byStep := byStep + 10;  END_IF

	40:	byStep := byStep + 10;

	50:(*Read if Feature was succesful R32 Read*)
		 IF usiState = 2#1010_0000 THEN
			(*Write Feature Register*)
			usiCtrl := byFeatureReg;
			usiCtrl.7 := TRUE;
			usiCtrl.6 := TRUE;
			iDataOut := iDataIn;(*Leave other settings*)
			CASE bySensorType OF
				0:	iDataOut.15 := FALSE;	iDataOut.14 := FALSE;	iDataOut.13 :=	FALSE;	iDataOut.12 := FALSE;(*PT1000*)
				1:	iDataOut.15 := FALSE;	iDataOut.14 := FALSE;	iDataOut.13 :=	FALSE;	iDataOut.12 := TRUE;(*NI1000*)
				2:	iDataOut.15 := FALSE;	iDataOut.14 := FALSE;	iDataOut.13 :=	TRUE;	iDataOut.12 := FALSE;(*RSNI1000*)
			ELSE
				bBusy := FALSE;
				bError := TRUE;
			END_CASE
		ELSE
				bBusy := FALSE;
				bError := TRUE;
		END_IF
		(* Jak nie ma bledy to dalej, jak blad to do kroku bledu *)
		IF bError THEN byStep := 255; ELSE byStep := byStep + 10;  END_IF

	60:	byStep := byStep + 10;(*Czekamy*)

	70:(*Read if Feature was succesful R32 Read*)
		 IF usiState = 2#1010_0000 THEN
			CASE byFurtherElements OF
			0: ; (* Nie zmieniamy parametru *)
			50..62, 100, 101, 200, 255: (* Wpisujemy odpowiednia wartosc do rejestru 39  *)
				usiCtrl := byFurtherElementsReg;
				usiCtrl.7 := TRUE;(*tryb register comm*)
				usiCtrl.6 := TRUE;(*true -zaspis rejestru, false - odczyt*)
				iDataOut := byFurtherElements;
			ELSE
				bBusy := FALSE;
				bError := TRUE;
			END_CASE
		ELSE
				bBusy := FALSE;
				bError := TRUE;
		END_IF

		(* Jak nie ma bledy to dalej, jak blad to do kroku bledu *)
		IF bError THEN byStep := 255; ELSE byStep := byStep + 10;  END_IF

	80:	byStep := byStep + 10;(*Czekamy*)

	90: 	 IF usiState = 2#1010_0000 OR usiState = 2#1010_0111  THEN (* R32 lub R39 *)
			(* Zamykamy rejestry *)
			usiCtrl := byCodeWordReg;
			usiCtrl.7 := TRUE;(*tryb register comm*)
			usiCtrl.6 := TRUE;(*true -zaspis rejestru, false - odczyt*)
			iDataOut := 0;
		ELSE
			bBusy := FALSE;
			bError := TRUE;
		END_IF
		(* Jak nie ma bledy to dalej, jak blad to do kroku bledu *)
		IF bError THEN byStep := 255; ELSE byStep := byStep + 10;  END_IF

	100: byStep := byStep + 10;(*Czekamy*)

	110: IF usiState = 2#10011111 THEN (* Zapisano 0 do R31 *)
			usiCtrl		:= 0;
			iDataOut 	:= 0;
			bBusy 		:= FALSE;
			bDone 		:= TRUE;
			byStep 		:= 0;
		END_IF
	255:	(*Error - proba zamkniecia rejestrow*)
		usiCtrl		:= byCodeWordReg;
		usiCtrl.7 	:= TRUE;
		usiCtrl.6 	:= TRUE;
		iDataOut 	:= 0;
		byStep 		:= 0;
END_CASE

END_FUNCTION_BLOCK

// ---- POUs/KL_Terminals/FB_KL32x8_1channelEx.TcPOU
(************************************************************************************************)
(*							Beckhoff Automation Poland											*)
(*							FB_KL32x8_1channelEx v1.0											*)
(*									17.07.2015													*)
(* 				-Dodane bDisableChannel															*)
(*		Blok funkcyjny konfigurujący kanał modułu KL32x8 dla określonego typu czujnika			*)
(*______________________________________________________________________________________________*)

FUNCTION_BLOCK FB_KL32x8_1channelEx
(*Objaśnienie procedur*)
(*	Control Byte
	BIT7 = 1 Register Mode
	BIT6 = 0 Read Register
	BIT6 = 1 Write Register
	BIT5-BIT0 -> Register Number
	
	usStatus BYTE
	BIT7 -> Writing Acknowledgement
	BIT5-BIT0 -> Which Register was Read
	
	R31 - CodeWord Register Code: 16#1235*)
VAR_INPUT
	bChange:				BOOL;	(*Rising edge activated function block*)
	bDisableChannel: 		BOOL; 	(* Disable the channel completely *)
	bySensorType:			BYTE;	(*Sensor type	R32 - Feature Register:
													BIT15	BIT14	BIT13	BIT12	Element	
								bySensorType = 0		0		0		0		0		PT1000
								bySensorType = 1		0		0		0		1		NI1000
								bySensorType = 2		0		0		1		0		RSNI1000*)
	byFurtherElements: 		BYTE; (* R39: Further elements (supported by KL3208-0010, from firmware version 1C and hardware version 01)
									  50 	NCT1K8			-40°C ... 130°C
									  51 	NCT1K8_TK		-30°C ... 150°C
									  52 	NCT2K2			-50°C ... 130°C
									  53 	NCT3K			-50°C ...   80°C
									  54 	NCT5K			-40°C ... 100°C
									  55 	NTC10K			-30°C ... 150°C
									  56 	NTC10KPRE		-30°C ... 150°C
									  57 	NTC10K_3204	-40°C ... 110°C
									  58 	NTC10KTYP2	-50°C ... 130°C
									  59 	NTC10KTYP3	-50°C ... 130°C
									  60 	NTC10KDALE	-50°C ... 130°C
									  61 	NTC10K3A221	-40°C ... 130°C
									  62 	NTC20K			-20°C ... 150°C
									100		Poti, resolution 0.1 Ohm	0 ... 5 kOhm
									101 	Poti, resolution 1 Ohm	0 ... 10 kOhm
									200 	NTC100K		-40°C ... 130°C
									255 	user defined NTC*)
	wR41: 					WORD;	(*B-Parameter for user defined NTC*)
	wR42: 					WORD; 	(*Resistance at 25°C for user defined NTC*)
	wR43: 					WORD; 	(*Reference temperature for user defined NTC*)
	wR44: 					WORD; 	(*Lower range limit for user defined NTC*)
	wR45: 					WORD; 	(*Upper range limit for user defined NTC*)
	usiState :				USINT;	(*Linked with KL32x8 - Channel X - Status*)
	iDataIn:				INT;	(*Linked with KL32x8 - Channel X - DataIn*)
END_VAR
VAR_OUTPUT
	bBusy: 					BOOL;	(* FB has job *)
	bDone:					BOOL;	(*If the execution of the function block is without error this output is set*)
	bError:					BOOL;	(*If an error is occur during the execution of the function block this output is set*)
	usiCtrl:				USINT;	(*Linked with KL32x8 - Channel X - Ctrl*)
	iDataOut:				INT;	(*Linked with KL32x8 - Channel X - DataOut*)
END_VAR
VAR
	byStep: 				BYTE;
	rtChange:				R_TRIG;
END_VAR
VAR CONSTANT
	byCodeWordReg: 			BYTE := 31;
	byFeatureReg: 			BYTE := 32;
	byFurtherElementsReg: 	BYTE := 39;
	wCodeWord:				WORD := 16#1235;
END_VAR

rtChange(CLK:= bChange);
IF rtChange.Q  THEN
	byStep := 10;
	bBusy := TRUE;
	bDone := FALSE;
	bError := FALSE;
END_IF
CASE byStep OF
	0:
		usiCtrl := 0;
		iDataOut := 0;

	10:	(*Write Code*)
		usiCtrl := byCodeWordReg;
		usiCtrl.7 := TRUE;(*tryb register comm*)
		usiCtrl.6 := TRUE;(*true -zaspis rejestru, false - odczyt*)
		iDataOut := WORD_TO_INT(wCodeWord);
		byStep := byStep + 10;

	20:	byStep := byStep + 10;(*czekamy*)

	30:	(*Read if Code write was succesful R31 Read*)
		IF usiState = 2#1001_1111 THEN
			(*Read Feature Register*)
			usiCtrl := byFeatureReg;
			usiCtrl.7 := TRUE;
			usiCtrl.6 := FALSE;
		ELSE
			bBusy := FALSE;
			bError := TRUE;
		END_IF
		(* Jak nie ma bledy to dalej, jak blad to do kroku bledu *)
		IF bError THEN byStep := 255; ELSE byStep := byStep + 10;  END_IF

	40:	byStep := byStep + 10;

	50:(*Read if Feature was succesful R32 Read*)
		 IF usiState = 2#1010_0000 THEN
			(*Write Feature Register*)
			usiCtrl := byFeatureReg;
			usiCtrl.7 := TRUE;
			usiCtrl.6 := TRUE;
			iDataOut := iDataIn;(*Leave other settings*)
			iDataOut.11 := bDisableChannel; (* Disable the channel completely *)
			CASE bySensorType OF
				0:	iDataOut.15 := FALSE;	iDataOut.14 := FALSE;	iDataOut.13 :=	FALSE;	iDataOut.12 := FALSE;(*PT1000*)
				1:	iDataOut.15 := FALSE;	iDataOut.14 := FALSE;	iDataOut.13 :=	FALSE;	iDataOut.12 := TRUE;(*NI1000*)
				2:	iDataOut.15 := FALSE;	iDataOut.14 := FALSE;	iDataOut.13 :=	TRUE;	iDataOut.12 := FALSE;(*RSNI1000*)
			ELSE
				bBusy := FALSE;
				bError := TRUE;
			END_CASE
		ELSE
				bBusy := FALSE;
				bError := TRUE;
		END_IF
		(* Jak nie ma bledy to dalej, jak blad to do kroku bledu *)
		IF bError THEN byStep := 255; ELSE byStep := byStep + 10;  END_IF

	60:	byStep := byStep + 10;(*Czekamy*)

	70:(*Read if Feature was succesful R32 Read*)
		 IF usiState = 2#1010_0000 THEN
			CASE byFurtherElements OF
			0, 50..62, 100, 101, 200, 255: (* Wpisujemy odpowiednia wartosc do rejestru 39  *)
				usiCtrl := byFurtherElementsReg;
				usiCtrl.7 := TRUE;(*tryb register comm*)
				usiCtrl.6 := TRUE;(*true -zaspis rejestru, false - odczyt*)
				iDataOut := byFurtherElements;
			ELSE
				bBusy := FALSE;
				bError := TRUE;
			END_CASE
		ELSE
				bBusy := FALSE;
				bError := TRUE;
		END_IF

		(* Jak nie ma bledy to dalej, jak blad to do kroku bledu *)
		IF bError THEN byStep := 255; ELSE byStep := byStep + 10;  END_IF

	80:	byStep := byStep + 10;(*Czekamy*)

	90: IF usiState = 2#1010_0111  THEN (* R39 zapisany prawidlowo *)
			usiCtrl := 2#10_1001; (* Zapis do rejestru 41 *)
			usiCtrl.7 := TRUE;(*tryb register comm*)
			usiCtrl.6 := TRUE;(*true -zaspis rejestru, false - odczyt*)
			iDataOut := WORD_TO_INT(wR41);
			byStep := byStep + 10;(*Dalej*)
		ELSE
			bBusy := FALSE;
			bError := TRUE;
			byStep := 255;(* Krok bledu *)
		END_IF

	100: byStep := byStep + 10;(*Czekamy*)

	110: IF usiState = 2#1010_1001  THEN (* R41 zapisany prawidlowo *)
			usiCtrl := 2#10_1010; (* Zapis do rejestru 42 *)
			usiCtrl.7 := TRUE;(*tryb register comm*)
			usiCtrl.6 := TRUE;(*true -zaspis rejestru, false - odczyt*)
			iDataOut := WORD_TO_INT(wR42);
			byStep := byStep + 10;(*Dalej*)
		ELSE
			bBusy := FALSE;
			bError := TRUE;
			byStep := 255;(* Krok bledu *)
		END_IF

	120: byStep := byStep + 10;(*Czekamy*)

	130: IF usiState = 2#1010_1010  THEN (* R42 zapisany prawidlowo *)
			usiCtrl := 2#10_1011; (* Zapis do rejestru 43 *)
			usiCtrl.7 := TRUE;(*tryb register comm*)
			usiCtrl.6 := TRUE;(*true -zaspis rejestru, false - odczyt*)
			iDataOut := WORD_TO_INT(wR43);
			byStep := byStep + 10;(*Dalej*)
		ELSE
			bBusy := FALSE;
			bError := TRUE;
			byStep := 255;(* Krok bledu *)
		END_IF

	140: byStep := byStep + 10;(*Czekamy*)

	150: IF usiState = 2#1010_1011  THEN (* R43 zapisany prawidlowo *)
			usiCtrl := 2#10_1100; (* Zapis do rejestru 44 *)
			usiCtrl.7 := TRUE;(*tryb register comm*)
			usiCtrl.6 := TRUE;(*true -zaspis rejestru, false - odczyt*)
			iDataOut := WORD_TO_INT(wR44);
			byStep := byStep + 10;(*Dalej*)
		ELSE
			bBusy := FALSE;
			bError := TRUE;
			byStep := 255;(* Krok bledu *)
		END_IF

	160: byStep := byStep + 10;(*Czekamy*)

	170: IF usiState = 2#1010_1100  THEN (* R44 zapisany prawidlowo *)
			usiCtrl := 2#10_1101; (* Zapis do rejestru 45 *)
			usiCtrl.7 := TRUE;(*tryb register comm*)
			usiCtrl.6 := TRUE;(*true -zaspis rejestru, false - odczyt*)
			iDataOut := word_to_int(wR45);
			byStep := byStep + 10;(*Dalej*)
		ELSE
			bBusy := FALSE;
			bError := TRUE;
			byStep := 255;(* Krok bledu *)
		END_IF

	180: byStep := byStep + 10;(*Czekamy*)

	190: IF usiState = 2#1010_1101  THEN (* R45 zapisany prawidlowo *)
			byStep := 200;(*Idz do zamkniecia rejestrow*)
		ELSE
			bBusy := FALSE;
			bError := TRUE;
			byStep := 255; (* Krok bledu *)
		END_IF

	200:(* Zamykamy rejestry *)
		usiCtrl := byCodeWordReg;
		usiCtrl.7 := TRUE;(*tryb register comm*)
		usiCtrl.6 := TRUE;(*true -zaspis rejestru, false - odczyt*)
		iDataOut := 0;
		byStep := byStep + 10;(*Czekamy*)

	210: byStep := byStep + 10;(*Czekamy*)

	220: IF usiState = 2#10011111 THEN (* Zapisano 0 do R31 *)
			usiCtrl		:= 0;
			iDataOut 	:= 0;
			bBusy 		:= FALSE;
			bDone 		:= TRUE;
			byStep 		:= 0;
		END_IF
	255:	(*Error - proba zamkniecia rejestrow*)
		usiCtrl		:= byCodeWordReg;
		usiCtrl.7 	:= TRUE;
		usiCtrl.6 	:= TRUE;
		iDataOut 	:= 0;
		byStep 		:= 0;
END_CASE

END_FUNCTION_BLOCK

// ---- POUs/KL_Terminals/FB_KL3403_1channel.TcPOU
(****************************************************************************************)
(*							Beckhoff Automation Poland									*)
(*								KL3403_1channel v1.2									*)
(*									03.11.2010											*)
(*					Blok funkcyjny zliczający wyświetlający parametry sieci.			*)
(*							Współpracuje z modułem KL3403.								*)
(*______________________________________________________________________________________*)

FUNCTION_BLOCK FB_KL3403_1channel
VAR_INPUT
	bEnable				:	BOOL;		(* Uruchomienie pomiarów*)
	bResetEnergy		:	BOOL; 		(* Narastające zbocze kasuje żużycie energii*)
END_VAR
VAR_OUTPUT
	wCurrentRMS			: 	WORD;		(* Natężenie prądu, rozdzielczość: 0.001A *)
	wVoltageRMS			: 	WORD;		(* Napięcie, rozdzielczość: 0.1V  *)
	wPower				:	WORD;		(* Moc, rozdzielczość: 0.1 W*)
	wCosFi				:	WORD;		(* cos Fi, rozdzielczość: 0.01 *)
	wEnergy				:	WORD;		(* Zużyta energia, rozdzielczość: 0.01 kWh*)
	bUndervoltage		: 	BOOL;		(* V_L1-N < R36 value*)
	bError				:	BOOL;		(* Błąd odczytu*)
	BProcDatIdx			:	BYTE;		(* Index aktualnie czytanych danych procesowych*)
END_VAR
VAR
	ibyState AT %I*		:	BYTE;		(* Płączone z  KL3403 - Channel X - State*)
	iwDataIn AT %I*		:	WORD;		(* Połączone z  KL3403 - Channel X - DataIn*)
	qbyCtrl AT %Q*		:	BYTE;		(* Połączone z KL3403 - Channel X - Ctrl*)
	qwDataOut AT %Q*	:	WORD;		(* Połączone z KL3403 - Channel X - DataOut*)

	BProcDatIdxChoose	:	BYTE;
	BProcDatIdxIs		:	BYTE;
	bAckPDM				:	BOOL;
	i					:	BYTE;
	imax				:	BYTE	:= 7;
	T1					:	TON;
	error1				:	BOOL;
	RisingEdge			:	R_TRIG;
	Step				:	INT;
	bMeasure			:	BOOL	:=TRUE;
END_VAR

(*Zerowanie energii*)
RisingEdge(CLK:= bResetEnergy);
IF RisingEdge.Q THEN bMeasure := FALSE; END_IF

IF bMeasure THEN
	(* wybor zmiennej pomierzonej lub wyliczonej do odczytu z rejestru DATA IN w KL3403
	    w ramach 'process image', zapis do zmiennej kontrolnej Ctrl typu BYTE *)
	qbyCtrl:=0;
	qbyCtrl:=BProcDatIdxChoose;

	(* odczyt potwierdzenia ze zmiennej STATE umieszczenia w rejestrze DATA IN zadanej zmiennej (prad, napiecie itp.)  *)
	BProcDatIdxIs:=0;
	BProcDatIdxIs:=2#00001111 AND ibyState;	(*change: V1.2*)
	BProcDatIdx:=BProcDatIdxIs;

	(*Acknowledgement for process data mode and Voltage between L1 and N less  than Undervoltage threshold *)
	bAckPDM:=ibyState.7;
	bUndervoltage:=ibyState.6;

	(* przepisanie opowiedniej zmiennej odczytanej z rejestru KL3403 po potwierdzeniu
	    umieszczenia jej w rejestrze DATA IN w KL3403 *)
	IF bEnable THEN
		IF i>imax THEN i:=0; END_IF;
		CASE i OF
			0:	BProcDatIdxChoose:=0;
			1:	BProcDatIdxChoose:=1;
			2:	BProcDatIdxChoose:=2;
			3:	BProcDatIdxChoose:=3;
			4:	BProcDatIdxChoose:=4;
			(*5:	BProcDatIdxChoose:=5;
			6:	BProcDatIdxChoose:=6;
			7:	BProcDatIdxChoose:=7;*)
		END_CASE;
		IF BProcDatIdxIs=BProcDatIdxChoose THEN
			CASE BProcDatIdxChoose OF
				0:	wCurrentRMS:=		iwDataIn;
				1:	wVoltageRMS:=		iwDataIn;
				2:	wPower:=			iwDataIn;
				3:	wCosFi:=			iwDataIn;
				4:	wEnergy:=			iwDataIn;
				(*5:	wPeakCurrent:=		wDataIn;
				6:	wPeakVoltage:=		wDataIn;
				7:	wPeakPower:=		wDataIn;*)
			END_CASE;
			i:=i+1;(*Odczyt następnej wartości*)
		END_IF;
	ELSE
	(*Gdy nie odczytujemy*)
		i:=0;
		BProcDatIdxChoose:=0;
	END_IF;

	(* obsluga bledow *)
	T1( IN:=error1 OR bAckPDM, PT:= T#500ms );
	IF BProcDatIdxChoose<>BProcDatIdxIs THEN
		error1:=TRUE;
	ELSE
		error1:=FALSE;
	END_IF;
	bError:=T1.Q;
ELSE
	CASE Step OF
	0:
	(*Czekamy*)
	IF  RisingEdge.Q THEN
		qbyCtrl:=2#11011111; (* otwieramy do zapisu R31*)
		qwDataOut:=16#1235; (* i wpisujemy 1235 hex*)
		Step:=Step+10;
	END_IF;

	10:
	IF ibyState=2#10011111  THEN
		(*Wpisujemy 16#1004 DO rejestru 7*)
		qbyCtrl:=199; (*1|1|Reg_No*)
		qwDataOut:=16#1004;
		Step:=Step+10;
	END_IF

	20:
	(* sprawdzamy, czy dobrze wpisalismy *)(*1|0|Reg_No*)
	IF ibyState=135 THEN
		qbyCtrl:=199; (*1|1|Reg_No*)
		qwDataOut:=0;
		Step:=Step+10;
	END_IF;

	30:

	IF ibyState.7=TRUE THEN
		qbyCtrl:=2#11011111; (* rejestr 31 wpisujemy wartosc 0*)
		qwDataOut:=0;
		Step:=Step+10;
	END_IF

	40:
	IF ibyState=2#10011111 THEN
		qbyCtrl.7:=0;(*zamykamy rejestr*)
		Step:=Step+10;
	END_IF

	50:
	IF ibyState.7=0 THEN
		Step:=0;
		bMeasure:=TRUE;
	END_IF

	END_CASE
END_IF

END_FUNCTION_BLOCK

// ---- POUs/KL_Terminals/FB_PowerMeasuring.TcPOU
(****************************************************************************************************)
(*							Beckhoff Automation Poland												*)
(*							FB_PowerMeasuring v1.3													*)
(*									24.05.2011														*)
(*			Blok funkcyjny zliczający zużycie energii. Współpracuje z modułem KL3403.				*)
(*			Konieczne jest dodanie biblioteki TcUtilities.lib, TcSystem.lib oraz TcBase.lib			*)
(*			Dane wyjściowe to raport roczny w formie tablicy 12 elementów typu ST_KL3403_Report		*)
(*				Summary: WORD; - całkowite zużycie energii = Tarrif1 + Tarrif2						*)
(*				SummaryPrice:WORD;- całkowity koszt energii = Tarrif1Price + Tarrif2Price			*)
(*				Tarrif1: WORD;																		*)
(*				Tarrif1Price:WORD;																	*)
(*				Tarrif2: WORD;																		*)
(*				Tarrif2Price:WORD;																	*)
(* 			Konieczne jest dodanie biblioteki TcUtilities.lib, TcSystem.lib oraz TcBase.lib			*)
(*		UWAGA!!!																					*)
(*		Blok ten korzysta z czasu systemowego, podawanego na wejście bloku.							*)
(*		Nie można wywoływać tego bloku bez podania czasu na wejściu,								*)
(*		ponieważ wówczas przyjmuje on wartości zerowe												*)
(*__________________________________________________________________________________________________*)

FUNCTION_BLOCK FB_PowerMeasuring
VAR_INPUT
	wValue: 			WORD; 			(*Zliczana wartość*)
	bTariff_Ex: 		BOOL; 			(*Sygnał droższej taryfy*)
	rFactor_1: 			REAL;	 		(*Współczynnik mnożący taryfy tańszej, w PLN*)
	rFactor_2: 			REAL;			(*Współczynnik mnożący taryfy droższej, w PLN*)
	strAktCzas:			TIMESTRUCT;		(*Aktualny czas w formie struktury*)
END_VAR
VAR_IN_OUT
	arrReport: 			ARRAY [1..12] OF ST_KL3403_Report;(*Raport z ostatnich 12 mesięcy*)
END_VAR
VAR
	wOldTariff1: 		WORD;		(*Wartość taryfy tańszej z bieżącego miesiąca*)
	wOldTariff2: 		WORD;		(*Wartość taryfy droższej z bieżącego miesiąca*)
	RisingEdge: 		R_TRIG;		(*Przełączenie na taryfę droższą*)
	FallingEdge: 		F_TRIG;		(*Przełączenie na taryfę tańszą*)
	wOldMonth: 			WORD; 		(*Poprzedni miesiąc*)
	wFreeze: 			WORD; 		(*Wartość w momencie przełączenia taryf*)
	bFirstCycle: 		BOOL:=TRUE;	(*Oznaczenie pierwszego cyklu programu*)
END_VAR

	(*Zapisanie początkowej wartości po restarcie programu*)
	IF bFirstCycle THEN
		(*Wpisanie aktualnych danych z pamięci nieulotnej*)
		wOldTariff1 := arrReport[strAktCzas.wMonth].Tarrif1;
		wOldTariff2 := arrReport[strAktCzas.wMonth].Tarrif2;
		(*Uzupełnienie wpisu o aktualnej wartości*)
		wFreeze := wValue;
		bFirstCycle := FALSE;
	END_IF
	(*Zapisanie początkowej wartości po restarcie modułu*)
	IF  wFreeze > wValue THEN
		wFreeze := wValue;
		wOldTariff1 := 0;
		wOldTariff2 := 0;
		arrReport[wOldMonth].Tarrif2 := 0;
		arrReport[wOldMonth].Tarrif1 := 0;
	END_IF

	(*Wykrycie przełączenia na taryfę tanią i obliczenie ostatniego przyrostu taryfy taniej*)
	RisingEdge(CLK:= bTariff_Ex);
	IF RisingEdge.Q THEN
		wOldTariff1 := wOldTariff1 + (wValue - wFreeze);
		wFreeze := wValue;
	END_IF
	(*Wykrycie przełączenia na taryfę drogą i obliczenie ostatniego przyrostu taryfy drogiej*)
	FallingEdge(CLK:= bTariff_Ex);
	IF FallingEdge.Q THEN
		wOldTariff2 := wOldTariff2 + (wValue - wFreeze);
		wFreeze := wValue;
	END_IF

	(*Sprawdzamy czy nadal mamy ten sam miesiąc*)
	IF strAktCzas.wMonth <> wOldMonth THEN
		(*Zapamiętanie stanów i wyzerowanie liczników w nowym miesiącu*)
		wOldMonth := strAktCzas.wMonth;
		wOldTariff1 := 0;
		wOldTariff2 := 0;
		wFreeze := wValue; (*Wartość przy przełączeniu taryf*)
	ELSE
		(*Uzupełnienie wpisów w tabeli*)
		IF bTariff_Ex THEN
			arrReport[wOldMonth].Tarrif2 := wOldTariff2 + (wValue-wFreeze);
			arrReport[wOldMonth].Tarrif2Price := REAL_TO_WORD((wOldTariff2 +wValue-wFreeze)* rFactor_2);
		ELSE
			arrReport[wOldMonth].Tarrif1 := wOldTariff1 + (wValue-wFreeze);
			arrReport[wOldMonth].Tarrif1Price := REAL_TO_WORD((wOldTariff1 + wValue-wFreeze)* rFactor_1);
		END_IF
		arrReport[wOldMonth].Summary := arrReport[wOldMonth].Tarrif1 + arrReport[wOldMonth].Tarrif2;
		arrReport[wOldMonth].SummaryPrice := arrReport[wOldMonth].Tarrif1Price + arrReport[wOldMonth].Tarrif2Price;
	END_IF;

END_FUNCTION_BLOCK

// ---- POUs/NC/FB_AX5000_Diag_MC2.TcPOU
(************************************************************************************************)
(*							Beckhoff Automation Poland											*)
(*							FB_AX5000_Diag_MC2  v1.0											*)
(*									24.5.2011													*)
(*			Blok funkcyjny czytający podstawowe parametry serwa AX5xxx i jego błedy				*)
(*				Odczytane dane wpisuje do zmiennej typu ST_AX5000_Diag_MC2						*)
(*______________________________________________________________________________________________*)
FUNCTION_BLOCK FB_AX5000_Diag_MC2
VAR_OUTPUT
	bError					:	BOOL;
	ST_DIAG					:	ST_AX5000_Diag_MC2;
END_VAR
VAR_IN_OUT
	Axis					:	Axis_REF;
END_VAR
VAR
	fb_ReadAmplifierTemp		:	FB_SoEReadAmplifierTemperature;		(*MC2Drive*)
	fb_ReadDCBusCurrent		:	FB_SoEReadDcBusCurrent;				(*MC2Drive*)
	fb_ReadDCBusVoltage		: 	FB_SoEReadDcBusVoltage;				(*MC2Drive*)
	fb_ReadMotorTemp			:	FB_SoEReadMotorTemperature;			(*MC2Drive*)
	fb_ReadDiagMessage		:	FB_SoEReadDiagMessage;				(*MC2Drive*)
	fb_DiagNumber			:	FB_SoEReadDiagNumber;				(*MC2Drive*)
	fb_ReadDiagList			:	FB_SoEReadDiagNumberList;			(*MC2Drive*)
	fb_ReadC1Diagnostic		:	FB_SoERead;

	timer					:	TON;
	DiagList				:	ST_SoE_DiagNumList;
	bFirstCycle				:	BOOL	:=TRUE;
	sDiagnosticMessage		:	ST_SoE_STRING;
	ft1						:	F_TRIG;
	ft2						:	F_TRIG;
	ft3						:	F_TRIG;
	ft4						:	F_TRIG;
	ft5						:	F_TRIG;
	ft6						:	F_TRIG;
	ft7						:	F_TRIG;
	Watchdog				:	TON;
	Delay					:	TP;
END_VAR
VAR // added by the converter: edge detectors and wires of the graphical bodies
    _w1, _w2 : BOOL;
    _w3, _w4, _w5, _w6, _w7, _w8 : ANY;
END_VAR

_w2 := _w1 OR bFirstCycle;
ft2(CLK := fb_ReadDCBusCurrent.Busy); // F_TRIG
fb_ReadMotorTemp(NetId := '', Execute := _w3, Timeout := T#1s, Axis := Axis); // FB_SoEReadMotorTemperature
ft3(CLK := fb_ReadMotorTemp.Busy); // F_TRIG
ST_DIAG.nMotor_Temp := fb_ReadMotorTemp.MotorTemperature;
ST_DIAG.sDiagnosticMessage := _w4;
fb_DiagNumber(NetId := '', Execute := _w5, Timeout := T#1s, Axis := Axis); // FB_SoEReadDiagNumber
ft5(CLK := fb_DiagNumber.Busy); // F_TRIG
_w6 := ft5.Q AND NOT fb_DiagNumber.Error;
fb_ReadDiagMessage(NetId := '', Execute := _w7, Timeout := T#1s, Axis := Axis); // FB_SoEReadDiagMessage
_w7 := ft3.Q AND NOT fb_ReadMotorTemp.Error;
ft4(CLK := fb_ReadDiagMessage.Busy); // F_TRIG
ST_DIAG.nDiagNumber := fb_DiagNumber.DiagNumber;
IF _w5 THEN _w4 := sDiagnosticMessage.strData; END_IF
sDiagnosticMessage := fb_ReadDiagMessage.DiagMessage;
_w5 := ft4.Q AND NOT fb_ReadDiagMessage.Error;
bFirstCycle R= fb_ReadAmplifierTemp.Busy;
ft1(CLK := fb_ReadAmplifierTemp.Busy); // F_TRIG
fb_ReadAmplifierTemp(NetId := '', Execute := _w2, Timeout := T#1s, Axis := Axis); // FB_SoEReadAmplifierTemperature
Watchdog(IN := NOT _w8, PT := T#10s); // TON
ST_DIAG.nDrive_Temp := fb_ReadAmplifierTemp.AmplifierTemperature;
Delay(IN := Watchdog.Q, PT := T#3s); // TP
bError := Watchdog.Q;
fb_ReadDCBusCurrent(NetId := '', Execute := _w8, Timeout := T#1s, Axis := Axis); // FB_SoEReadDcBusCurrent
bFirstCycle S= Delay.Q;
ST_DIAG.nDC_Bus_Current := fb_ReadDCBusCurrent.DcBusCurrent;
fb_ReadDCBusVoltage(
    NetId := '',
    Execute := ft2.Q AND NOT fb_ReadDCBusCurrent.Error,
    Timeout := T#1s,
    Axis := Axis); // FB_SoEReadDcBusVoltage
_w8 := ft1.Q AND NOT fb_ReadAmplifierTemp.Error;
_w3 := ft3.Q AND NOT fb_ReadDCBusVoltage.Error;
ft3(CLK := fb_ReadDCBusVoltage.Busy); // F_TRIG
ST_DIAG.nMotor_Temp := fb_ReadDCBusVoltage.DcBusVoltage;
fb_ReadDiagList(
    NetId := '',
    Execute := _w6,
    Timeout := T#1s,
    pDiagNumber := ADR(ST_DIAG.DiagList),
    Size := SIZEOF(ST_DIAG.DiagList),
    Axis := Axis); // FB_SoEReadDiagNumberList
ft6(CLK := fb_ReadDiagList.Busy); // F_TRIG
fb_ReadC1Diagnostic(
    NetId := '',
    Idn := 11,
    Element := 16#40,
    pDstBuf := ADR(ST_DIAG.DiagList),
    BufLen := SIZEOF(ST_DIAG.DiagList),
    Execute := ft6.Q AND NOT fb_ReadDiagList.Error,
    Timeout := T#1s,
    Axis := Axis); // FB_SoERead
ft7(CLK := fb_ReadC1Diagnostic.Busy); // F_TRIG
_w1 := ft7.Q AND NOT fb_ReadC1Diagnostic.Error;

END_FUNCTION_BLOCK

// ---- POUs/NC/FB_AxisParameter.TcPOU
//==================================================================================================
//					Beckhoff Automation Poland
//							30.05.2017
//		Blok funkcyjny zmieniajacy krańcówki SW górną i dolną
// 	v1.0 	|| TC v 3.1.4020.32 	|| - pierwsza wersja
//==================================================================================================
FUNCTION_BLOCK FB_AxisParameter
VAR_INPUT
	udiAxisID				: UDINT;		// ID osi
	bRead					: BOOL;
	bWrite					: BOOL;
	bReset					: BOOL; // Not yet
// Set values
	lrSetMinPos				: LREAL;
	lrSetMaxPos				: LREAL;
	bSetMinMon				: BOOL;
	bSetMaxMon				: BOOL;
END_VAR
VAR_OUTPUT
	//	
	bBusy					: BOOL;
	bError					: BOOL;
	udiErrorID				: UDINT;
// Actual values	
	lrActMinPos				: LREAL;
	lrActMaxPos				: LREAL;
	bActMinMon				: BOOL;
	bActMaxMon				: BOOL;
END_VAR
VAR
	iStepWrite				: INT;
	iStepRead				: INT;
	wSetMinMon				: WORD;
	wSetMaxMon				: WORD;
	wActMinMon				: WORD;
	wActMaxMon				: WORD;
// FBs
	rtRead					: R_TRIG;
	rtWrite					: R_TRIG;
	fbADSREAD				: ADSREAD;
	fbADSWRITE				: ADSWRITE;
END_VAR
VAR CONSTANT
	udiIDXGRP_OFFS			: UDINT := 16#0000_5000;
	udiIDXOFFS_MinMon		: UDINT := 16#0000_000B;	// 2B
	udiIDXOFFS_MinPos		: UDINT := 16#0000_000D;	// 8B
	udiIDXOFFS_MaxMon		: UDINT := 16#0000_000C;	// 2B	
	udiIDXOFFS_MaxPos		: UDINT := 16#0000_000E;	// 8B
END_VAR

// Triggery
rtRead(CLK:= bRead, Q=> );
rtWrite(CLK:= bWrite, Q=> );

ACT_ReadParams();
ACT_WriteParams();	

	
// Read parameters
	fbADSREAD(	NETID:= '', 
				PORT:= 500,
				IDXGRP:= udiIDXGRP_OFFS + udiAxisID);
	
// Write parameters
	fbADSWRITE(	NETID:= '', 
				PORT:= 500,
				IDXGRP:= udiIDXGRP_OFFS + udiAxisID);

ACTION ACT_ReadParams:
CASE iStepRead OF

0: // Idle
	IF rtRead.Q AND NOT bBusy THEN
		bBusy 					:= TRUE;
		bError 					:= FALSE;
		udiErrorID				:= 0;
		// MinMon 16#0000_000B;	// 2B
		fbADSREAD.READ			:= TRUE;
		fbADSREAD.IDXOFFS		:= 16#0000_000B;
		fbADSREAD.LEN			:= 2;
		fbADSREAD.DESTADDR		:= ADR(wActMinMon);
		iStepRead				:= iStepRead + 5;
	END_IF
	
5, 15, 25: // Wait CMD for end
	fbADSREAD.READ				:= FALSE;
	IF NOT fbADSREAD.BUSY AND NOT fbADSREAD.ERR THEN
		iStepRead				:= iStepRead + 5;
	ELSIF fbADSREAD.ERR THEN
		iStepRead				:= 1000;
	END_IF
	
10: // udiIDXOFFS_MinPos		: UDINT := 16#0000_000D;	// 8B
	fbADSREAD.READ				:= TRUE;
	fbADSREAD.IDXOFFS			:= 16#0000_000D;
	fbADSREAD.LEN				:= 8;
	fbADSREAD.DESTADDR			:= ADR(lrActMinPos);
	iStepRead					:= iStepRead + 5;

20: // 	udiIDXOFFS_MaxMon		: UDINT := 16#0000_000C;	// 2B
	fbADSREAD.READ				:= TRUE;
	fbADSREAD.IDXOFFS			:= 16#0000_000C;
	fbADSREAD.LEN				:= 2;
	fbADSREAD.DESTADDR			:= ADR(wActMaxMon);
	iStepRead					:= iStepRead + 5;

30: // 		udiIDXOFFS_MaxPos		: UDINT := 16#0000_000E;	// 8B
	fbADSREAD.READ				:= TRUE;
	fbADSREAD.IDXOFFS			:= 16#0000_000E;
	fbADSREAD.LEN				:= 8;
	fbADSREAD.DESTADDR			:= ADR(lrActMaxPos);
	iStepRead					:= iStepRead + 5;
		
35: // 	End
	fbADSREAD.READ				:= FALSE;
	IF NOT fbADSREAD.BUSY AND NOT fbADSREAD.ERR THEN
		bActMinMon				:= wActMinMon.0;
		bActMaxMon				:= wActMaxMon.0;
		bBusy 					:= FALSE;
		iStepRead				:= 0;
	ELSIF fbADSREAD.ERR THEN
		iStepRead				:= 1000;
	END_IF
	
1000:
	bBusy 						:= FALSE;
	bError 						:= TRUE;
	udiErrorID					:= fbADSREAD.ERRID;
	iStepRead					:= 0;

END_CASE
END_ACTION

ACTION ACT_WriteParams:
CASE iStepWrite OF

0: // Idle
	IF rtWrite.Q AND NOT bBusy THEN
		bBusy 					:= TRUE;
		bError 					:= FALSE;
		udiErrorID				:= 0;
		// MinMon 16#0000_000B;	// 2B
		wSetMinMon.0 			:= bSetMinMon;
		fbADSWRITE.WRITE		:= TRUE;
		fbADSWRITE.IDXOFFS		:= 16#0000_000B;
		fbADSWRITE.LEN			:= 2;
		fbADSWRITE.SRCADDR		:= ADR(wSetMinMon);
		iStepWrite				:= iStepWrite + 5;
	END_IF
	
5, 15, 25: // Wait CMD for end
	fbADSWRITE.WRITE			:= FALSE;
	IF NOT fbADSWRITE.BUSY AND NOT fbADSWRITE.ERR THEN
		iStepWrite				:= iStepWrite + 5;
	ELSIF fbADSWRITE.ERR THEN
		iStepWrite				:= 1000;
	END_IF
	
10: // udiIDXOFFS_MinPos		: UDINT := 16#0000_000D;	// 8B
	fbADSWRITE.WRITE			:= TRUE;
	fbADSWRITE.IDXOFFS			:= 16#0000_000D;
	fbADSWRITE.LEN				:= 8;
	fbADSWRITE.SRCADDR			:= ADR(lrSetMinPos);
	iStepWrite					:= iStepWrite + 5;

20: // 	udiIDXOFFS_MaxMon		: UDINT := 16#0000_000C;	// 2B
	wSetMaxMon.0 				:= bSetMaxMon;
	fbADSWRITE.WRITE			:= TRUE;
	fbADSWRITE.IDXOFFS			:= 16#0000_000C;
	fbADSWRITE.LEN				:= 2;
	fbADSWRITE.SRCADDR			:= ADR(wSetMaxMon);
	iStepWrite					:= iStepWrite + 5;

